(* CODESYS project mobject-converters.library
   Company: mobject
   DefaultNamespace: mobject-converters
   Version: 1.0.2
   Placeholder: mobject-converters
   Author: mobject dev team
   Title: mobject-converters

Project tree, tasks and I/O mapping:
  libraries: Tc2_System, * (Beckhoff Automation GmbH); mobject-constants-datatype-limits, 1.0.0 (mobject)
  Converters/
    BOOL_TO_/
      function TryConvert_BOOL_TO_BOOL [ST]
      function TryConvert_BOOL_TO_BYTE [ST]
      function TryConvert_BOOL_TO_DATE [ST]
      function TryConvert_BOOL_TO_Destination [ST]
      function TryConvert_BOOL_TO_DINT [ST]
      function TryConvert_BOOL_TO_DT [ST]
      function TryConvert_BOOL_TO_DWORD [ST]
      function TryConvert_BOOL_TO_INT [ST]
      function TryConvert_BOOL_TO_LINT [ST]
      function TryConvert_BOOL_TO_LREAL [ST]
      function TryConvert_BOOL_TO_LWORD [ST]
      function TryConvert_BOOL_TO_REAL [ST]
      function TryConvert_BOOL_TO_SINT [ST]
      function TryConvert_BOOL_TO_STRING [ST]
      function TryConvert_BOOL_TO_TIME [ST]
      function TryConvert_BOOL_TO_TOD [ST]
      function TryConvert_BOOL_TO_UDINT [ST]
      function TryConvert_BOOL_TO_UINT [ST]
      function TryConvert_BOOL_TO_ULINT [ST]
      function TryConvert_BOOL_TO_USINT [ST]
      function TryConvert_BOOL_TO_WORD [ST]
    BYTE_TO_/
      function TryConvert_BYTE_TO_BOOL [ST]
      function TryConvert_BYTE_TO_BYTE [ST]
      function TryConvert_BYTE_TO_DATE [ST]
      function TryConvert_BYTE_TO_Destination [ST]
      function TryConvert_BYTE_TO_DINT [ST]
      function TryConvert_BYTE_TO_DT [ST]
      function TryConvert_BYTE_TO_DWORD [ST]
      function TryConvert_BYTE_TO_INT [ST]
      function TryConvert_BYTE_TO_LINT [ST]
      function TryConvert_BYTE_TO_LREAL [ST]
      function TryConvert_BYTE_TO_LWORD [ST]
      function TryConvert_BYTE_TO_REAL [ST]
      function TryConvert_BYTE_TO_SINT [ST]
      function TryConvert_BYTE_TO_STRING [ST]
      function TryConvert_BYTE_TO_TIME [ST]
      function TryConvert_BYTE_TO_TOD [ST]
      function TryConvert_BYTE_TO_UDINT [ST]
      function TryConvert_BYTE_TO_UINT [ST]
      function TryConvert_BYTE_TO_ULINT [ST]
      function TryConvert_BYTE_TO_USINT [ST]
      function TryConvert_BYTE_TO_WORD [ST]
    DATE_TO_/
      function TryConvert_DATE_TO_BOOL [ST]
      function TryConvert_DATE_TO_BYTE [ST]
      function TryConvert_DATE_TO_DATE [ST]
      function TryConvert_DATE_TO_Destination [ST]
      function TryConvert_DATE_TO_DINT [ST]
      function TryConvert_DATE_TO_DT [ST]
      function TryConvert_DATE_TO_DWORD [ST]
      function TryConvert_DATE_TO_INT [ST]
      function TryConvert_DATE_TO_LINT [ST]
      function TryConvert_DATE_TO_LREAL [ST]
      function TryConvert_DATE_TO_LWORD [ST]
      function TryConvert_DATE_TO_REAL [ST]
      function TryConvert_DATE_TO_SINT [ST]
      function TryConvert_DATE_TO_STRING [ST]
      function TryConvert_DATE_TO_TIME [ST]
      function TryConvert_DATE_TO_TOD [ST]
      function TryConvert_DATE_TO_UDINT [ST]
      function TryConvert_DATE_TO_UINT [ST]
      function TryConvert_DATE_TO_ULINT [ST]
      function TryConvert_DATE_TO_USINT [ST]
      function TryConvert_DATE_TO_WORD [ST]
    DINT_TO_/
      function TryConvert_DINT_TO_BOOL [ST]
      function TryConvert_DINT_TO_BYTE [ST]
      function TryConvert_DINT_TO_DATE [ST]
      function TryConvert_DINT_TO_Destination [ST]
      function TryConvert_DINT_TO_DINT [ST]
      function TryConvert_DINT_TO_DT [ST]
      function TryConvert_DINT_TO_DWORD [ST]
      function TryConvert_DINT_TO_INT [ST]
      function TryConvert_DINT_TO_LINT [ST]
      function TryConvert_DINT_TO_LREAL [ST]
      function TryConvert_DINT_TO_LWORD [ST]
      function TryConvert_DINT_TO_REAL [ST]
      function TryConvert_DINT_TO_SINT [ST]
      function TryConvert_DINT_TO_STRING [ST]
      function TryConvert_DINT_TO_TIME [ST]
      function TryConvert_DINT_TO_TOD [ST]
      function TryConvert_DINT_TO_UDINT [ST]
      function TryConvert_DINT_TO_UINT [ST]
      function TryConvert_DINT_TO_ULINT [ST]
      function TryConvert_DINT_TO_USINT [ST]
      function TryConvert_DINT_TO_WORD [ST]
    DT_TO_/
      function TryConvert_DT_TO_BOOL [ST]
      function TryConvert_DT_TO_BYTE [ST]
      function TryConvert_DT_TO_DATE [ST]
      function TryConvert_DT_TO_Destination [ST]
      function TryConvert_DT_TO_DINT [ST]
      function TryConvert_DT_TO_DT [ST]
      function TryConvert_DT_TO_DWORD [ST]
      function TryConvert_DT_TO_INT [ST]
      function TryConvert_DT_TO_LINT [ST]
      function TryConvert_DT_TO_LREAL [ST]
      function TryConvert_DT_TO_LWORD [ST]
      function TryConvert_DT_TO_REAL [ST]
      function TryConvert_DT_TO_SINT [ST]
      function TryConvert_DT_TO_STRING [ST]
      function TryConvert_DT_TO_TIME [ST]
      function TryConvert_DT_TO_TOD [ST]
      function TryConvert_DT_TO_UDINT [ST]
      function TryConvert_DT_TO_UINT [ST]
      function TryConvert_DT_TO_ULINT [ST]
      function TryConvert_DT_TO_USINT [ST]
      function TryConvert_DT_TO_WORD [ST]
    DWORD_TO_/
      function TryConvert_DWORD_TO_BOOL [ST]
      function TryConvert_DWORD_TO_BYTE [ST]
      function TryConvert_DWORD_TO_DATE [ST]
      function TryConvert_DWORD_TO_Destination [ST]
      function TryConvert_DWORD_TO_DINT [ST]
      function TryConvert_DWORD_TO_DT [ST]
      function TryConvert_DWORD_TO_DWORD [ST]
      function TryConvert_DWORD_TO_INT [ST]
      function TryConvert_DWORD_TO_LINT [ST]
      function TryConvert_DWORD_TO_LREAL [ST]
      function TryConvert_DWORD_TO_LWORD [ST]
      function TryConvert_DWORD_TO_REAL [ST]
      function TryConvert_DWORD_TO_SINT [ST]
      function TryConvert_DWORD_TO_STRING [ST]
      function TryConvert_DWORD_TO_TIME [ST]
      function TryConvert_DWORD_TO_TOD [ST]
      function TryConvert_DWORD_TO_UDINT [ST]
      function TryConvert_DWORD_TO_UINT [ST]
      function TryConvert_DWORD_TO_ULINT [ST]
      function TryConvert_DWORD_TO_USINT [ST]
      function TryConvert_DWORD_TO_WORD [ST]
    INT_TO_/
      function TryConvert_INT_TO_BOOL [ST]
      function TryConvert_INT_TO_BYTE [ST]
      function TryConvert_INT_TO_DATE [ST]
      function TryConvert_INT_TO_Destination [ST]
      function TryConvert_INT_TO_DINT [ST]
      function TryConvert_INT_TO_DT [ST]
      function TryConvert_INT_TO_DWORD [ST]
      function TryConvert_INT_TO_INT [ST]
      function TryConvert_INT_TO_LINT [ST]
      function TryConvert_INT_TO_LREAL [ST]
      function TryConvert_INT_TO_LWORD [ST]
      function TryConvert_INT_TO_REAL [ST]
      function TryConvert_INT_TO_SINT [ST]
      function TryConvert_INT_TO_STRING [ST]
      function TryConvert_INT_TO_TIME [ST]
      function TryConvert_INT_TO_TOD [ST]
      function TryConvert_INT_TO_UDINT [ST]
      function TryConvert_INT_TO_UINT [ST]
      function TryConvert_INT_TO_ULINT [ST]
      function TryConvert_INT_TO_USINT [ST]
      function TryConvert_INT_TO_WORD [ST]
    LINT_TO_/
      function TryConvert_LINT_TO_BOOL [ST]
      function TryConvert_LINT_TO_BYTE [ST]
      function TryConvert_LINT_TO_DATE [ST]
      function TryConvert_LINT_TO_Destination [ST]
      function TryConvert_LINT_TO_DINT [ST]
      function TryConvert_LINT_TO_DT [ST]
      function TryConvert_LINT_TO_DWORD [ST]
      function TryConvert_LINT_TO_INT [ST]
      function TryConvert_LINT_TO_LINT [ST]
      function TryConvert_LINT_TO_LREAL [ST]
      function TryConvert_LINT_TO_LWORD [ST]
      function TryConvert_LINT_TO_REAL [ST]
      function TryConvert_LINT_TO_SINT [ST]
      function TryConvert_LINT_TO_STRING [ST]
      function TryConvert_LINT_TO_TIME [ST]
      function TryConvert_LINT_TO_TOD [ST]
      function TryConvert_LINT_TO_UDINT [ST]
      function TryConvert_LINT_TO_UINT [ST]
      function TryConvert_LINT_TO_ULINT [ST]
      function TryConvert_LINT_TO_USINT [ST]
      function TryConvert_LINT_TO_WORD [ST]
    LREAL_TO_/
      function TryConvert_LREAL_TO_BOOL [ST]
      function TryConvert_LREAL_TO_BYTE [ST]
      function TryConvert_LREAL_TO_DATE [ST]
      function TryConvert_LREAL_TO_Destination [ST]
      function TryConvert_LREAL_TO_DINT [ST]
      function TryConvert_LREAL_TO_DT [ST]
      function TryConvert_LREAL_TO_DWORD [ST]
      function TryConvert_LREAL_TO_INT [ST]
      function TryConvert_LREAL_TO_LINT [ST]
      function TryConvert_LREAL_TO_LREAL [ST]
      function TryConvert_LREAL_TO_LWORD [ST]
      function TryConvert_LREAL_TO_REAL [ST]
      function TryConvert_LREAL_TO_SINT [ST]
      function TryConvert_LREAL_TO_STRING [ST]
      function TryConvert_LREAL_TO_TIME [ST]
      function TryConvert_LREAL_TO_TOD [ST]
      function TryConvert_LREAL_TO_UDINT [ST]
      function TryConvert_LREAL_TO_UINT [ST]
      function TryConvert_LREAL_TO_ULINT [ST]
      function TryConvert_LREAL_TO_USINT [ST]
      function TryConvert_LREAL_TO_WORD [ST]
    LWORD_TO_/
      function TryConvert_LWORD_TO_BOOL [ST]
      function TryConvert_LWORD_TO_BYTE [ST]
      function TryConvert_LWORD_TO_DATE [ST]
      function TryConvert_LWORD_TO_Destination [ST]
      function TryConvert_LWORD_TO_DINT [ST]
      function TryConvert_LWORD_TO_DT [ST]
      function TryConvert_LWORD_TO_DWORD [ST]
      function TryConvert_LWORD_TO_INT [ST]
      function TryConvert_LWORD_TO_LINT [ST]
      function TryConvert_LWORD_TO_LREAL [ST]
      function TryConvert_LWORD_TO_LWORD [ST]
      function TryConvert_LWORD_TO_REAL [ST]
      function TryConvert_LWORD_TO_SINT [ST]
      function TryConvert_LWORD_TO_STRING [ST]
      function TryConvert_LWORD_TO_TIME [ST]
      function TryConvert_LWORD_TO_TOD [ST]
      function TryConvert_LWORD_TO_UDINT [ST]
      function TryConvert_LWORD_TO_UINT [ST]
      function TryConvert_LWORD_TO_ULINT [ST]
      function TryConvert_LWORD_TO_USINT [ST]
      function TryConvert_LWORD_TO_WORD [ST]
    REAL_TO_/
      function TryConvert_REAL_TO_BOOL [ST]
      function TryConvert_REAL_TO_BYTE [ST]
      function TryConvert_REAL_TO_DATE [ST]
      function TryConvert_REAL_TO_Destination [ST]
      function TryConvert_REAL_TO_DINT [ST]
      function TryConvert_REAL_TO_DT [ST]
      function TryConvert_REAL_TO_DWORD [ST]
      function TryConvert_REAL_TO_INT [ST]
      function TryConvert_REAL_TO_LINT [ST]
      function TryConvert_REAL_TO_LREAL [ST]
      function TryConvert_REAL_TO_LWORD [ST]
      function TryConvert_REAL_TO_REAL [ST]
      function TryConvert_REAL_TO_SINT [ST]
      function TryConvert_REAL_TO_STRING [ST]
      function TryConvert_REAL_TO_TIME [ST]
      function TryConvert_REAL_TO_TOD [ST]
      function TryConvert_REAL_TO_UDINT [ST]
      function TryConvert_REAL_TO_UINT [ST]
      function TryConvert_REAL_TO_ULINT [ST]
      function TryConvert_REAL_TO_USINT [ST]
      function TryConvert_REAL_TO_WORD [ST]
    SINT_TO_/
      function TryConvert_SINT_TO_BOOL [ST]
      function TryConvert_SINT_TO_BYTE [ST]
      function TryConvert_SINT_TO_DATE [ST]
      function TryConvert_SINT_TO_Destination [ST]
      function TryConvert_SINT_TO_DINT [ST]
      function TryConvert_SINT_TO_DT [ST]
      function TryConvert_SINT_TO_DWORD [ST]
      function TryConvert_SINT_TO_INT [ST]
      function TryConvert_SINT_TO_LINT [ST]
      function TryConvert_SINT_TO_LREAL [ST]
      function TryConvert_SINT_TO_LWORD [ST]
      function TryConvert_SINT_TO_REAL [ST]
      function TryConvert_SINT_TO_SINT [ST]
      function TryConvert_SINT_TO_STRING [ST]
      function TryConvert_SINT_TO_TIME [ST]
      function TryConvert_SINT_TO_TOD [ST]
      function TryConvert_SINT_TO_UDINT [ST]
      function TryConvert_SINT_TO_UINT [ST]
      function TryConvert_SINT_TO_ULINT [ST]
      function TryConvert_SINT_TO_USINT [ST]
      function TryConvert_SINT_TO_WORD [ST]
    STRING_TO_/
      function TryConvert_STRING_TO_BOOL [ST]
      function TryConvert_STRING_TO_BYTE [ST]
      function TryConvert_STRING_TO_DATE [ST]
      function TryConvert_STRING_TO_Destination [ST]
      function TryConvert_STRING_TO_DINT [ST]
      function TryConvert_STRING_TO_DT [ST]
      function TryConvert_STRING_TO_DWORD [ST]
      function TryConvert_STRING_TO_INT [ST]
      function TryConvert_STRING_TO_LINT [ST]
      function TryConvert_STRING_TO_LREAL [ST]
      function TryConvert_STRING_TO_LWORD [ST]
      function TryConvert_STRING_TO_REAL [ST]
      function TryConvert_STRING_TO_SINT [ST]
      function TryConvert_STRING_TO_STRING [ST]
      function TryConvert_STRING_TO_TIME [ST]
      function TryConvert_STRING_TO_TOD [ST]
      function TryConvert_STRING_TO_UDINT [ST]
      function TryConvert_STRING_TO_UINT [ST]
      function TryConvert_STRING_TO_ULINT [ST]
      function TryConvert_STRING_TO_USINT [ST]
      function TryConvert_STRING_TO_WORD [ST]
    TIME_TO_/
      function TryConvert_TIME_TO_BOOL [ST]
      function TryConvert_TIME_TO_BYTE [ST]
      function TryConvert_TIME_TO_DATE [ST]
      function TryConvert_TIME_TO_Destination [ST]
      function TryConvert_TIME_TO_DINT [ST]
      function TryConvert_TIME_TO_DT [ST]
      function TryConvert_TIME_TO_DWORD [ST]
      function TryConvert_TIME_TO_INT [ST]
      function TryConvert_TIME_TO_LINT [ST]
      function TryConvert_TIME_TO_LREAL [ST]
      function TryConvert_TIME_TO_LWORD [ST]
      function TryConvert_TIME_TO_REAL [ST]
      function TryConvert_TIME_TO_SINT [ST]
      function TryConvert_TIME_TO_STRING [ST]
      function TryConvert_TIME_TO_TIME [ST]
      function TryConvert_TIME_TO_TOD [ST]
      function TryConvert_TIME_TO_UDINT [ST]
      function TryConvert_TIME_TO_UINT [ST]
      function TryConvert_TIME_TO_ULINT [ST]
      function TryConvert_TIME_TO_USINT [ST]
      function TryConvert_TIME_TO_WORD [ST]
    TOD_TO_/
      function TryConvert_TOD_TO_BOOL [ST]
      function TryConvert_TOD_TO_BYTE [ST]
      function TryConvert_TOD_TO_DATE [ST]
      function TryConvert_TOD_TO_Destination [ST]
      function TryConvert_TOD_TO_DINT [ST]
      function TryConvert_TOD_TO_DT [ST]
      function TryConvert_TOD_TO_DWORD [ST]
      function TryConvert_TOD_TO_INT [ST]
      function TryConvert_TOD_TO_LINT [ST]
      function TryConvert_TOD_TO_LREAL [ST]
      function TryConvert_TOD_TO_LWORD [ST]
      function TryConvert_TOD_TO_REAL [ST]
      function TryConvert_TOD_TO_SINT [ST]
      function TryConvert_TOD_TO_STRING [ST]
      function TryConvert_TOD_TO_TIME [ST]
      function TryConvert_TOD_TO_TOD [ST]
      function TryConvert_TOD_TO_UDINT [ST]
      function TryConvert_TOD_TO_UINT [ST]
      function TryConvert_TOD_TO_ULINT [ST]
      function TryConvert_TOD_TO_USINT [ST]
      function TryConvert_TOD_TO_WORD [ST]
    UDINT_TO_/
      function TryConvert_UDINT_TO_BOOL [ST]
      function TryConvert_UDINT_TO_BYTE [ST]
      function TryConvert_UDINT_TO_DATE [ST]
      function TryConvert_UDINT_TO_Destination [ST]
      function TryConvert_UDINT_TO_DINT [ST]
      function TryConvert_UDINT_TO_DT [ST]
      function TryConvert_UDINT_TO_DWORD [ST]
      function TryConvert_UDINT_TO_INT [ST]
      function TryConvert_UDINT_TO_LINT [ST]
      function TryConvert_UDINT_TO_LREAL [ST]
      function TryConvert_UDINT_TO_LWORD [ST]
      function TryConvert_UDINT_TO_REAL [ST]
      function TryConvert_UDINT_TO_SINT [ST]
      function TryConvert_UDINT_TO_STRING [ST]
      function TryConvert_UDINT_TO_TIME [ST]
      function TryConvert_UDINT_TO_TOD [ST]
      function TryConvert_UDINT_TO_UDINT [ST]
      function TryConvert_UDINT_TO_UINT [ST]
      function TryConvert_UDINT_TO_ULINT [ST]
      function TryConvert_UDINT_TO_USINT [ST]
      function TryConvert_UDINT_TO_WORD [ST]
    UINT_TO_/
      function TryConvert_UINT_TO_BOOL [ST]
      function TryConvert_UINT_TO_BYTE [ST]
      function TryConvert_UINT_TO_DATE [ST]
      function TryConvert_UINT_TO_Destination [ST]
      function TryConvert_UINT_TO_DINT [ST]
      function TryConvert_UINT_TO_DT [ST]
      function TryConvert_UINT_TO_DWORD [ST]
      function TryConvert_UINT_TO_INT [ST]
      function TryConvert_UINT_TO_LINT [ST]
      function TryConvert_UINT_TO_LREAL [ST]
      function TryConvert_UINT_TO_LWORD [ST]
      function TryConvert_UINT_TO_REAL [ST]
      function TryConvert_UINT_TO_SINT [ST]
      function TryConvert_UINT_TO_STRING [ST]
      function TryConvert_UINT_TO_TIME [ST]
      function TryConvert_UINT_TO_TOD [ST]
      function TryConvert_UINT_TO_UDINT [ST]
      function TryConvert_UINT_TO_UINT [ST]
      function TryConvert_UINT_TO_ULINT [ST]
      function TryConvert_UINT_TO_USINT [ST]
      function TryConvert_UINT_TO_WORD [ST]
    ULINT_TO_/
      function TryConvert_ULINT_TO_BOOL [ST]
      function TryConvert_ULINT_TO_BYTE [ST]
      function TryConvert_ULINT_TO_DATE [ST]
      function TryConvert_ULINT_TO_Destination [ST]
      function TryConvert_ULINT_TO_DINT [ST]
      function TryConvert_ULINT_TO_DT [ST]
      function TryConvert_ULINT_TO_DWORD [ST]
      function TryConvert_ULINT_TO_INT [ST]
      function TryConvert_ULINT_TO_LINT [ST]
      function TryConvert_ULINT_TO_LREAL [ST]
      function TryConvert_ULINT_TO_LWORD [ST]
      function TryConvert_ULINT_TO_REAL [ST]
      function TryConvert_ULINT_TO_SINT [ST]
      function TryConvert_ULINT_TO_STRING [ST]
      function TryConvert_ULINT_TO_TIME [ST]
      function TryConvert_ULINT_TO_TOD [ST]
      function TryConvert_ULINT_TO_UDINT [ST]
      function TryConvert_ULINT_TO_UINT [ST]
      function TryConvert_ULINT_TO_ULINT [ST]
      function TryConvert_ULINT_TO_USINT [ST]
      function TryConvert_ULINT_TO_WORD [ST]
    USINT_TO_/
      function TryConvert_USINT_TO_BOOL [ST]
      function TryConvert_USINT_TO_BYTE [ST]
      function TryConvert_USINT_TO_DATE [ST]
      function TryConvert_USINT_TO_Destination [ST]
      function TryConvert_USINT_TO_DINT [ST]
      function TryConvert_USINT_TO_DT [ST]
      function TryConvert_USINT_TO_DWORD [ST]
      function TryConvert_USINT_TO_INT [ST]
      function TryConvert_USINT_TO_LINT [ST]
      function TryConvert_USINT_TO_LREAL [ST]
      function TryConvert_USINT_TO_LWORD [ST]
      function TryConvert_USINT_TO_REAL [ST]
      function TryConvert_USINT_TO_SINT [ST]
      function TryConvert_USINT_TO_STRING [ST]
      function TryConvert_USINT_TO_TIME [ST]
      function TryConvert_USINT_TO_TOD [ST]
      function TryConvert_USINT_TO_UDINT [ST]
      function TryConvert_USINT_TO_UINT [ST]
      function TryConvert_USINT_TO_ULINT [ST]
      function TryConvert_USINT_TO_USINT [ST]
      function TryConvert_USINT_TO_WORD [ST]
    WORD_TO_/
      function TryConvert_WORD_TO_BOOL [ST]
      function TryConvert_WORD_TO_BYTE [ST]
      function TryConvert_WORD_TO_DATE [ST]
      function TryConvert_WORD_TO_Destination [ST]
      function TryConvert_WORD_TO_DINT [ST]
      function TryConvert_WORD_TO_DT [ST]
      function TryConvert_WORD_TO_DWORD [ST]
      function TryConvert_WORD_TO_INT [ST]
      function TryConvert_WORD_TO_LINT [ST]
      function TryConvert_WORD_TO_LREAL [ST]
      function TryConvert_WORD_TO_LWORD [ST]
      function TryConvert_WORD_TO_REAL [ST]
      function TryConvert_WORD_TO_SINT [ST]
      function TryConvert_WORD_TO_STRING [ST]
      function TryConvert_WORD_TO_TIME [ST]
      function TryConvert_WORD_TO_TOD [ST]
      function TryConvert_WORD_TO_UDINT [ST]
      function TryConvert_WORD_TO_UINT [ST]
      function TryConvert_WORD_TO_ULINT [ST]
      function TryConvert_WORD_TO_USINT [ST]
      function TryConvert_WORD_TO_WORD [ST]
    function TryConvert_Source_TO_Destination [ST]
*)

// Converters/BOOL_TO_/TryConvert_BOOL_TO_BOOL
FUNCTION TryConvert_BOOL_TO_BOOL : BOOL
VAR_INPUT
	in : BOOL;
	out : REFERENCE TO BOOL;
END_VAR

out := in;
TryConvert_BOOL_TO_BOOL := TRUE;

END_FUNCTION

// Converters/BOOL_TO_/TryConvert_BOOL_TO_BYTE
FUNCTION TryConvert_BOOL_TO_BYTE : BOOL
VAR_INPUT
	in : BOOL;
	out : REFERENCE TO BYTE;
END_VAR

out := BOOL_TO_BYTE(in);
TryConvert_BOOL_TO_BYTE := TRUE;

END_FUNCTION

// Converters/BOOL_TO_/TryConvert_BOOL_TO_DATE
FUNCTION TryConvert_BOOL_TO_DATE : BOOL
VAR_INPUT
	in : BOOL;
	out : REFERENCE TO DATE;
END_VAR

out := BOOL_TO_DATE(in);
TryConvert_BOOL_TO_DATE := TRUE;

END_FUNCTION

// Converters/BOOL_TO_/TryConvert_BOOL_TO_Destination
FUNCTION TryConvert_BOOL_TO_Destination : BOOL
VAR_INPUT
	in : BOOL;
	out : ANY;
END_VAR
VAR
	convertResult : BOOL := FALSE;
	convertAddress : PVOID;
	_BOOL : BOOL;
	_BYTE : BYTE;
	_WORD : WORD;
	_DWORD : DWORD;
	_LWORD : LWORD;
	_SINT : SINT;
	_INT : INT;
	_DINT : DINT;
	_LINT : LINT;
	_USINT : USINT;
	_UINT : UINT;
	_UDINT : UDINT;
	_ULINT : ULINT;
	_REAL : REAL;
	_LREAL : LREAL;
	_TIME : TIME;
	_TOD : TOD;
	_DATE : DATE;
	_DT : DT;
	_STRING : STRING;
END_VAR

CASE out.TypeClass OF
	__SYSTEM.TYPE_CLASS.TYPE_BOOL:
	
	convertResult := TryConvert_BOOL_TO_BOOL(in, _BOOL);
	IF convertResult THEN
		convertAddress := ADR(_BOOL);
	END_IF
	
	__SYSTEM.TYPE_CLASS.TYPE_BYTE:
	
	convertResult := TryConvert_BOOL_TO_BYTE(in, _BYTE);
	IF convertResult THEN
		convertAddress := ADR(_BYTE);
	END_IF
	
	__SYSTEM.TYPE_CLASS.TYPE_WORD:
	
	convertResult := TryConvert_BOOL_TO_WORD(in, _WORD);
	IF convertResult THEN
		convertAddress := ADR(_WORD);
	END_IF
	
	__SYSTEM.TYPE_CLASS.TYPE_DWORD:
	
	convertResult := TryConvert_BOOL_TO_DWORD(in, _DWORD);
	IF convertResult THEN
		convertAddress := ADR(_DWORD);
	END_IF
	
	__SYSTEM.TYPE_CLASS.TYPE_LWORD:
	
	convertResult := TryConvert_BOOL_TO_LWORD(in, _LWORD);
	IF convertResult THEN
		convertAddress := ADR(_LWORD);
	END_IF
	
	__SYSTEM.TYPE_CLASS.TYPE_SINT:
	
	convertResult := TryConvert_BOOL_TO_SINT(in, _SINT);
	IF convertResult THEN
		convertAddress := ADR(_SINT);
	END_IF
	
	__SYSTEM.TYPE_CLASS.TYPE_INT:
	
	convertResult := TryConvert_BOOL_TO_INT(in, _INT);
	IF convertResult THEN
		convertAddress := ADR(_INT);
	END_IF
	
	__SYSTEM.TYPE_CLASS.TYPE_DINT:
	
	convertResult := TryConvert_BOOL_TO_DINT(in, _DINT);
	IF convertResult THEN
		convertAddress := ADR(_DINT);
	END_IF
	
	__SYSTEM.TYPE_CLASS.TYPE_LINT:
	
	convertResult := TryConvert_BOOL_TO_LINT(in, _LINT);
	IF convertResult THEN
		convertAddress := ADR(_LINT);
	END_IF
	
	__SYSTEM.TYPE_CLASS.TYPE_USINT:
	
	convertResult := TryConvert_BOOL_TO_USINT(in, _USINT);
	IF convertResult THEN
		convertAddress := ADR(_USINT);
	END_IF
	
	__SYSTEM.TYPE_CLASS.TYPE_UINT:
	
	convertResult := TryConvert_BOOL_TO_UINT(in, _UINT);
	IF convertResult THEN
		convertAddress := ADR(_UINT);
	END_IF
	
	__SYSTEM.TYPE_CLASS.TYPE_UDINT:
	
	convertResult := TryConvert_BOOL_TO_UDINT(in, _UDINT);
	IF convertResult THEN
		convertAddress := ADR(_UDINT);
	END_IF
	
	__SYSTEM.TYPE_CLASS.TYPE_ULINT:
	
	convertResult := TryConvert_BOOL_TO_ULINT(in, _ULINT);
	IF convertResult THEN
		convertAddress := ADR(_ULINT);
	END_IF
	
	__SYSTEM.TYPE_CLASS.TYPE_REAL:
	
	convertResult := TryConvert_BOOL_TO_REAL(in, _REAL);
	IF convertResult THEN
		convertAddress := ADR(_REAL);
	END_IF
	
	__SYSTEM.TYPE_CLASS.TYPE_LREAL:
	
	convertResult := TryConvert_BOOL_TO_LREAL(in, _LREAL);
	IF convertResult THEN
		convertAddress := ADR(_LREAL);
	END_IF
	
	__SYSTEM.TYPE_CLASS.TYPE_TIME:
	
	convertResult := TryConvert_BOOL_TO_TIME(in, _TIME);
	IF convertResult THEN
		convertAddress := ADR(_TIME);
	END_IF
	
	__SYSTEM.TYPE_CLASS.TYPE_TIMEOFDAY:
	
	convertResult := TryConvert_BOOL_TO_TOD(in, _TOD);
	IF convertResult THEN
		convertAddress := ADR(_TOD);
	END_IF
	
	__SYSTEM.TYPE_CLASS.TYPE_DATE:
	
	convertResult := TryConvert_BOOL_TO_DATE(in, _DATE);
	IF convertResult THEN
		convertAddress := ADR(_DATE);
	END_IF
	
	__SYSTEM.TYPE_CLASS.TYPE_DATEANDTIME:
	
	convertResult := TryConvert_BOOL_TO_DT(in, _DT);
	IF convertResult THEN
		convertAddress := ADR(_DT);
	END_IF
	
	__SYSTEM.TYPE_CLASS.TYPE_STRING:
	
	convertResult := TryConvert_BOOL_TO_STRING(in, _STRING);
	IF convertResult THEN
		convertAddress := ADR(_STRING);
	END_IF
	
END_CASE

IF convertResult THEN
	memcpy(out.pValue,convertAddress,DINT_TO_UDINT(out.diSize));
END_IF

TryConvert_BOOL_TO_Destination := convertResult;

END_FUNCTION

// Converters/BOOL_TO_/TryConvert_BOOL_TO_WORD
FUNCTION TryConvert_BOOL_TO_WORD : BOOL
VAR_INPUT
	in : BOOL;
	out : REFERENCE TO WORD;
END_VAR

out := BOOL_TO_WORD(in);
TryConvert_BOOL_TO_WORD := TRUE;

END_FUNCTION

// Converters/BOOL_TO_/TryConvert_BOOL_TO_DWORD
FUNCTION TryConvert_BOOL_TO_DWORD : BOOL
VAR_INPUT
	in : BOOL;
	out : REFERENCE TO DWORD;
END_VAR

out := BOOL_TO_DWORD(in);
TryConvert_BOOL_TO_DWORD := TRUE;

END_FUNCTION

// Converters/BOOL_TO_/TryConvert_BOOL_TO_LWORD
FUNCTION TryConvert_BOOL_TO_LWORD : BOOL
VAR_INPUT
	in : BOOL;
	out : REFERENCE TO LWORD;
END_VAR

out := BOOL_TO_LWORD(in);
TryConvert_BOOL_TO_LWORD := TRUE;

END_FUNCTION

// Converters/BOOL_TO_/TryConvert_BOOL_TO_SINT
FUNCTION TryConvert_BOOL_TO_SINT : BOOL
VAR_INPUT
	in : BOOL;
	out : REFERENCE TO SINT;
END_VAR

out := BOOL_TO_SINT(in);
TryConvert_BOOL_TO_SINT := TRUE;

END_FUNCTION

// Converters/BOOL_TO_/TryConvert_BOOL_TO_INT
FUNCTION TryConvert_BOOL_TO_INT : BOOL
VAR_INPUT
	in : BOOL;
	out : REFERENCE TO INT;
END_VAR

out := BOOL_TO_INT(in);
TryConvert_BOOL_TO_INT := TRUE;

END_FUNCTION

// Converters/BOOL_TO_/TryConvert_BOOL_TO_DINT
FUNCTION TryConvert_BOOL_TO_DINT : BOOL
VAR_INPUT
	in : BOOL;
	out : REFERENCE TO DINT;
END_VAR

out := BOOL_TO_DINT(in);
TryConvert_BOOL_TO_DINT := TRUE;

END_FUNCTION

// Converters/BOOL_TO_/TryConvert_BOOL_TO_LINT
FUNCTION TryConvert_BOOL_TO_LINT : BOOL
VAR_INPUT
	in : BOOL;
	out : REFERENCE TO LINT;
END_VAR

out := BOOL_TO_LINT(in);
TryConvert_BOOL_TO_LINT := TRUE;

END_FUNCTION

// Converters/BOOL_TO_/TryConvert_BOOL_TO_USINT
FUNCTION TryConvert_BOOL_TO_USINT : BOOL
VAR_INPUT
	in : BOOL;
	out : REFERENCE TO USINT;
END_VAR

out := BOOL_TO_USINT(in);
TryConvert_BOOL_TO_USINT := TRUE;

END_FUNCTION

// Converters/BOOL_TO_/TryConvert_BOOL_TO_UINT
FUNCTION TryConvert_BOOL_TO_UINT : BOOL
VAR_INPUT
	in : BOOL;
	out : REFERENCE TO UINT;
END_VAR

out := BOOL_TO_UINT(in);
TryConvert_BOOL_TO_UINT := TRUE;

END_FUNCTION

// Converters/BOOL_TO_/TryConvert_BOOL_TO_UDINT
FUNCTION TryConvert_BOOL_TO_UDINT : BOOL
VAR_INPUT
	in : BOOL;
	out : REFERENCE TO UDINT;
END_VAR

out := BOOL_TO_UDINT(in);
TryConvert_BOOL_TO_UDINT := TRUE;

END_FUNCTION

// Converters/BOOL_TO_/TryConvert_BOOL_TO_ULINT
FUNCTION TryConvert_BOOL_TO_ULINT : BOOL
VAR_INPUT
	in : BOOL;
	out : REFERENCE TO ULINT;
END_VAR

out := BOOL_TO_ULINT(in);
TryConvert_BOOL_TO_ULINT := TRUE;

END_FUNCTION

// Converters/BOOL_TO_/TryConvert_BOOL_TO_REAL
FUNCTION TryConvert_BOOL_TO_REAL : BOOL
VAR_INPUT
	in : BOOL;
	out : REFERENCE TO REAL;
END_VAR

out := BOOL_TO_REAL(in);
TryConvert_BOOL_TO_REAL := TRUE;

END_FUNCTION

// Converters/BOOL_TO_/TryConvert_BOOL_TO_LREAL
FUNCTION TryConvert_BOOL_TO_LREAL : BOOL
VAR_INPUT
	in : BOOL;
	out : REFERENCE TO LREAL;
END_VAR

out := BOOL_TO_LREAL(in);
TryConvert_BOOL_TO_LREAL := TRUE;

END_FUNCTION

// Converters/BOOL_TO_/TryConvert_BOOL_TO_TIME
FUNCTION TryConvert_BOOL_TO_TIME : BOOL
VAR_INPUT
	in : BOOL;
	out : REFERENCE TO TIME;
END_VAR

out := BOOL_TO_TIME(in);
TryConvert_BOOL_TO_TIME := TRUE;

END_FUNCTION

// Converters/BOOL_TO_/TryConvert_BOOL_TO_TOD
FUNCTION TryConvert_BOOL_TO_TOD : BOOL
VAR_INPUT
	in : BOOL;
	out : REFERENCE TO TOD;
END_VAR

out := BOOL_TO_TOD(in);
TryConvert_BOOL_TO_TOD := TRUE;

END_FUNCTION

// Converters/BOOL_TO_/TryConvert_BOOL_TO_DT
FUNCTION TryConvert_BOOL_TO_DT : BOOL
VAR_INPUT
	in : BOOL;
	out : REFERENCE TO DT;
END_VAR

out := BOOL_TO_DT(in);
TryConvert_BOOL_TO_DT := TRUE;

END_FUNCTION

// Converters/BOOL_TO_/TryConvert_BOOL_TO_STRING
FUNCTION TryConvert_BOOL_TO_STRING : BOOL
VAR_INPUT
	in : BOOL;
	out : REFERENCE TO STRING;
END_VAR

out := BOOL_TO_STRING(in);
TryConvert_BOOL_TO_STRING := TRUE;

END_FUNCTION

// Converters/BYTE_TO_/TryConvert_BYTE_TO_BOOL
FUNCTION TryConvert_BYTE_TO_BOOL : BOOL
VAR_INPUT
	in : BYTE;
	out : REFERENCE TO BOOL;
END_VAR

out := BYTE_TO_BOOL(in);
TryConvert_BYTE_TO_BOOL := TRUE;

END_FUNCTION

// Converters/BYTE_TO_/TryConvert_BYTE_TO_BYTE
FUNCTION TryConvert_BYTE_TO_BYTE : BOOL
VAR_INPUT
	in : BYTE;
	out : REFERENCE TO BYTE;
END_VAR

out := in;
TryConvert_BYTE_TO_BYTE := TRUE;

END_FUNCTION

// Converters/BYTE_TO_/TryConvert_BYTE_TO_DATE
FUNCTION TryConvert_BYTE_TO_DATE : BOOL
VAR_INPUT
	in : BYTE;
	out : REFERENCE TO DATE;
END_VAR

out := BYTE_TO_DATE(in);
TryConvert_BYTE_TO_DATE := TRUE;

END_FUNCTION

// Converters/BYTE_TO_/TryConvert_BYTE_TO_Destination
FUNCTION TryConvert_BYTE_TO_Destination : BOOL
VAR_INPUT
	in : BYTE;
	out : ANY;
END_VAR
VAR
	convertResult : BOOL := FALSE;
	convertAddress : PVOID;
	_BOOL : BOOL;
	_BYTE : BYTE;
	_WORD : WORD;
	_DWORD : DWORD;
	_LWORD : LWORD;
	_SINT : SINT;
	_INT : INT;
	_DINT : DINT;
	_LINT : LINT;
	_USINT : USINT;
	_UINT : UINT;
	_UDINT : UDINT;
	_ULINT : ULINT;
	_REAL : REAL;
	_LREAL : LREAL;
	_TIME : TIME;
	_TOD : TOD;
	_DATE : DATE;
	_DT : DT;
	_STRING : STRING;
END_VAR

CASE out.TypeClass OF
	__SYSTEM.TYPE_CLASS.TYPE_BOOL:
	
	convertResult := TryConvert_BYTE_TO_BOOL(in, _BOOL);
	IF convertResult THEN
		convertAddress := ADR(_BOOL);
	END_IF
	
	__SYSTEM.TYPE_CLASS.TYPE_BYTE:
	
	convertResult := TryConvert_BYTE_TO_BYTE(in, _BYTE);
	IF convertResult THEN
		convertAddress := ADR(_BYTE);
	END_IF
	
	__SYSTEM.TYPE_CLASS.TYPE_WORD:
	
	convertResult := TryConvert_BYTE_TO_WORD(in, _WORD);
	IF convertResult THEN
		convertAddress := ADR(_WORD);
	END_IF
	
	__SYSTEM.TYPE_CLASS.TYPE_DWORD:
	
	convertResult := TryConvert_BYTE_TO_DWORD(in, _DWORD);
	IF convertResult THEN
		convertAddress := ADR(_DWORD);
	END_IF
	
	__SYSTEM.TYPE_CLASS.TYPE_LWORD:
	
	convertResult := TryConvert_BYTE_TO_LWORD(in, _LWORD);
	IF convertResult THEN
		convertAddress := ADR(_LWORD);
	END_IF
	
	__SYSTEM.TYPE_CLASS.TYPE_SINT:
	
	convertResult := TryConvert_BYTE_TO_SINT(in, _SINT);
	IF convertResult THEN
		convertAddress := ADR(_SINT);
	END_IF
	
	__SYSTEM.TYPE_CLASS.TYPE_INT:
	
	convertResult := TryConvert_BYTE_TO_INT(in, _INT);
	IF convertResult THEN
		convertAddress := ADR(_INT);
	END_IF
	
	__SYSTEM.TYPE_CLASS.TYPE_DINT:
	
	convertResult := TryConvert_BYTE_TO_DINT(in, _DINT);
	IF convertResult THEN
		convertAddress := ADR(_DINT);
	END_IF
	
	__SYSTEM.TYPE_CLASS.TYPE_LINT:
	
	convertResult := TryConvert_BYTE_TO_LINT(in, _LINT);
	IF convertResult THEN
		convertAddress := ADR(_LINT);
	END_IF
	
	__SYSTEM.TYPE_CLASS.TYPE_USINT:
	
	convertResult := TryConvert_BYTE_TO_USINT(in, _USINT);
	IF convertResult THEN
		convertAddress := ADR(_USINT);
	END_IF
	
	__SYSTEM.TYPE_CLASS.TYPE_UINT:
	
	convertResult := TryConvert_BYTE_TO_UINT(in, _UINT);
	IF convertResult THEN
		convertAddress := ADR(_UINT);
	END_IF
	
	__SYSTEM.TYPE_CLASS.TYPE_UDINT:
	
	convertResult := TryConvert_BYTE_TO_UDINT(in, _UDINT);
	IF convertResult THEN
		convertAddress := ADR(_UDINT);
	END_IF
	
	__SYSTEM.TYPE_CLASS.TYPE_ULINT:
	
	convertResult := TryConvert_BYTE_TO_ULINT(in, _ULINT);
	IF convertResult THEN
		convertAddress := ADR(_ULINT);
	END_IF
	
	__SYSTEM.TYPE_CLASS.TYPE_REAL:
	
	convertResult := TryConvert_BYTE_TO_REAL(in, _REAL);
	IF convertResult THEN
		convertAddress := ADR(_REAL);
	END_IF
	
	__SYSTEM.TYPE_CLASS.TYPE_LREAL:
	
	convertResult := TryConvert_BYTE_TO_LREAL(in, _LREAL);
	IF convertResult THEN
		convertAddress := ADR(_LREAL);
	END_IF
	
	__SYSTEM.TYPE_CLASS.TYPE_TIME:
	
	convertResult := TryConvert_BYTE_TO_TIME(in, _TIME);
	IF convertResult THEN
		convertAddress := ADR(_TIME);
	END_IF
	
	__SYSTEM.TYPE_CLASS.TYPE_TIMEOFDAY:
	
	convertResult := TryConvert_BYTE_TO_TOD(in, _TOD);
	IF convertResult THEN
		convertAddress := ADR(_TOD);
	END_IF
	
	__SYSTEM.TYPE_CLASS.TYPE_DATE:
	
	convertResult := TryConvert_BYTE_TO_DATE(in, _DATE);
	IF convertResult THEN
		convertAddress := ADR(_DATE);
	END_IF
	
	__SYSTEM.TYPE_CLASS.TYPE_DATEANDTIME:
	
	convertResult := TryConvert_BYTE_TO_DT(in, _DT);
	IF convertResult THEN
		convertAddress := ADR(_DT);
	END_IF
	
	__SYSTEM.TYPE_CLASS.TYPE_STRING:
	
	convertResult := TryConvert_BYTE_TO_STRING(in, _STRING);
	IF convertResult THEN
		convertAddress := ADR(_STRING);
	END_IF
	
END_CASE

IF convertResult THEN
	memcpy(out.pValue,convertAddress,DINT_TO_UDINT(out.diSize));
END_IF

TryConvert_BYTE_TO_Destination := convertResult;

END_FUNCTION

// Converters/BYTE_TO_/TryConvert_BYTE_TO_WORD
FUNCTION TryConvert_BYTE_TO_WORD : BOOL
VAR_INPUT
	in : BYTE;
	out : REFERENCE TO WORD;
END_VAR

out := BYTE_TO_WORD(in);
TryConvert_BYTE_TO_WORD := TRUE;

END_FUNCTION

// Converters/BYTE_TO_/TryConvert_BYTE_TO_DWORD
FUNCTION TryConvert_BYTE_TO_DWORD : BOOL
VAR_INPUT
	in : BYTE;
	out : REFERENCE TO DWORD;
END_VAR

out := BYTE_TO_DWORD(in);
TryConvert_BYTE_TO_DWORD := TRUE;

END_FUNCTION

// Converters/BYTE_TO_/TryConvert_BYTE_TO_LWORD
FUNCTION TryConvert_BYTE_TO_LWORD : BOOL
VAR_INPUT
	in : BYTE;
	out : REFERENCE TO LWORD;
END_VAR

out := BYTE_TO_LWORD(in);
TryConvert_BYTE_TO_LWORD := TRUE;

END_FUNCTION

// Converters/BYTE_TO_/TryConvert_BYTE_TO_SINT
FUNCTION TryConvert_BYTE_TO_SINT : BOOL
VAR_INPUT
	in : BYTE;
	out : REFERENCE TO SINT;
END_VAR

IF in > DatatypeLimits.MAX_VALUE_OF_BYTE_WHICH_CAN_BE_HELD_IN_A_SINT THEN
	RETURN;
END_IF

out := BYTE_TO_SINT(in);
TryConvert_BYTE_TO_SINT := TRUE;

END_FUNCTION

// Converters/BYTE_TO_/TryConvert_BYTE_TO_INT
FUNCTION TryConvert_BYTE_TO_INT : BOOL
VAR_INPUT
	in : BYTE;
	out : REFERENCE TO INT;
END_VAR

out := BYTE_TO_INT(in);
TryConvert_BYTE_TO_INT := TRUE;

END_FUNCTION

// Converters/BYTE_TO_/TryConvert_BYTE_TO_DINT
FUNCTION TryConvert_BYTE_TO_DINT : BOOL
VAR_INPUT
	in : BYTE;
	out : REFERENCE TO DINT;
END_VAR

out := BYTE_TO_DINT(in);
TryConvert_BYTE_TO_DINT := TRUE;

END_FUNCTION

// Converters/BYTE_TO_/TryConvert_BYTE_TO_LINT
FUNCTION TryConvert_BYTE_TO_LINT : BOOL
VAR_INPUT
	in : BYTE;
	out : REFERENCE TO LINT;
END_VAR

out := BYTE_TO_LINT(in);
TryConvert_BYTE_TO_LINT := TRUE;

END_FUNCTION

// Converters/BYTE_TO_/TryConvert_BYTE_TO_USINT
FUNCTION TryConvert_BYTE_TO_USINT : BOOL
VAR_INPUT
	in : BYTE;
	out : REFERENCE TO USINT;
END_VAR

out := BYTE_TO_USINT(in);
TryConvert_BYTE_TO_USINT := TRUE;

END_FUNCTION

// Converters/BYTE_TO_/TryConvert_BYTE_TO_UINT
FUNCTION TryConvert_BYTE_TO_UINT : BOOL
VAR_INPUT
	in : BYTE;
	out : REFERENCE TO UINT;
END_VAR

out := BYTE_TO_UINT(in);
TryConvert_BYTE_TO_UINT := TRUE;

END_FUNCTION

// Converters/BYTE_TO_/TryConvert_BYTE_TO_UDINT
FUNCTION TryConvert_BYTE_TO_UDINT : BOOL
VAR_INPUT
	in : BYTE;
	out : REFERENCE TO UDINT;
END_VAR

out := BYTE_TO_UDINT(in);
TryConvert_BYTE_TO_UDINT := TRUE;

END_FUNCTION

// Converters/BYTE_TO_/TryConvert_BYTE_TO_ULINT
FUNCTION TryConvert_BYTE_TO_ULINT : BOOL
VAR_INPUT
	in : BYTE;
	out : REFERENCE TO ULINT;
END_VAR

out := BYTE_TO_ULINT(in);
TryConvert_BYTE_TO_ULINT := TRUE;

END_FUNCTION

// Converters/BYTE_TO_/TryConvert_BYTE_TO_REAL
FUNCTION TryConvert_BYTE_TO_REAL : BOOL
VAR_INPUT
	in : BYTE;
	out : REFERENCE TO REAL;
END_VAR

out := BYTE_TO_REAL(in);
TryConvert_BYTE_TO_REAL := TRUE;

END_FUNCTION

// Converters/BYTE_TO_/TryConvert_BYTE_TO_LREAL
FUNCTION TryConvert_BYTE_TO_LREAL : BOOL
VAR_INPUT
	in : BYTE;
	out : REFERENCE TO LREAL;
END_VAR

out := BYTE_TO_LREAL(in);
TryConvert_BYTE_TO_LREAL := TRUE;

END_FUNCTION

// Converters/BYTE_TO_/TryConvert_BYTE_TO_TIME
FUNCTION TryConvert_BYTE_TO_TIME : BOOL
VAR_INPUT
	in : BYTE;
	out : REFERENCE TO TIME;
END_VAR

out := BYTE_TO_TIME(in);
TryConvert_BYTE_TO_TIME := TRUE;

END_FUNCTION

// Converters/BYTE_TO_/TryConvert_BYTE_TO_TOD
FUNCTION TryConvert_BYTE_TO_TOD : BOOL
VAR_INPUT
	in : BYTE;
	out : REFERENCE TO TOD;
END_VAR

out := BYTE_TO_TOD(in);
TryConvert_BYTE_TO_TOD := TRUE;

END_FUNCTION

// Converters/BYTE_TO_/TryConvert_BYTE_TO_DT
FUNCTION TryConvert_BYTE_TO_DT : BOOL
VAR_INPUT
	in : BYTE;
	out : REFERENCE TO DT;
END_VAR

out := BYTE_TO_DT(in);
TryConvert_BYTE_TO_DT := TRUE;

END_FUNCTION

// Converters/BYTE_TO_/TryConvert_BYTE_TO_STRING
FUNCTION TryConvert_BYTE_TO_STRING : BOOL
VAR_INPUT
	in : BYTE;
	out : REFERENCE TO STRING;
END_VAR

out := BYTE_TO_STRING(in);
TryConvert_BYTE_TO_STRING := TRUE;

END_FUNCTION

// Converters/DATE_TO_/TryConvert_DATE_TO_BOOL
FUNCTION TryConvert_DATE_TO_BOOL : BOOL
VAR_INPUT
	in : DATE;
	out : REFERENCE TO BOOL;
END_VAR

out := DATE_TO_BOOL(in);
TryConvert_DATE_TO_BOOL := TRUE;

END_FUNCTION

// Converters/DATE_TO_/TryConvert_DATE_TO_BYTE
FUNCTION TryConvert_DATE_TO_BYTE : BOOL
VAR_INPUT
	in : DATE;
	out : REFERENCE TO BYTE;
END_VAR

IF in > DatatypeLimits.MAX_VALUE_OF_DATE_WHICH_CAN_BE_HELD_IN_A_BYTE THEN
	RETURN;
END_IF

out := DATE_TO_BYTE(in);
TryConvert_DATE_TO_BYTE := TRUE;

END_FUNCTION

// Converters/DATE_TO_/TryConvert_DATE_TO_DATE
FUNCTION TryConvert_DATE_TO_DATE : BOOL
VAR_INPUT
	in : DATE;
	out : REFERENCE TO DATE;
END_VAR

out := in;
TryConvert_DATE_TO_DATE := TRUE;

END_FUNCTION

// Converters/DATE_TO_/TryConvert_DATE_TO_Destination
FUNCTION TryConvert_DATE_TO_Destination : BOOL
VAR_INPUT
	in : DATE;
	out : ANY;
END_VAR
VAR
	convertResult : BOOL := FALSE;
	convertAddress : PVOID;
	_BOOL : BOOL;
	_BYTE : BYTE;
	_WORD : WORD;
	_DWORD : DWORD;
	_LWORD : LWORD;
	_SINT : SINT;
	_INT : INT;
	_DINT : DINT;
	_LINT : LINT;
	_USINT : USINT;
	_UINT : UINT;
	_UDINT : UDINT;
	_ULINT : ULINT;
	_REAL : REAL;
	_LREAL : LREAL;
	_TIME : TIME;
	_TOD : TOD;
	_DATE : DATE;
	_DT : DT;
	_STRING : STRING;
END_VAR

CASE out.TypeClass OF
	__SYSTEM.TYPE_CLASS.TYPE_BOOL:
	
	convertResult := TryConvert_DATE_TO_BOOL(in, _BOOL);
	IF convertResult THEN
		convertAddress := ADR(_BOOL);
	END_IF
	
	__SYSTEM.TYPE_CLASS.TYPE_BYTE:
	
	convertResult := TryConvert_DATE_TO_BYTE(in, _BYTE);
	IF convertResult THEN
		convertAddress := ADR(_BYTE);
	END_IF
	
	__SYSTEM.TYPE_CLASS.TYPE_WORD:
	
	convertResult := TryConvert_DATE_TO_WORD(in, _WORD);
	IF convertResult THEN
		convertAddress := ADR(_WORD);
	END_IF
	
	__SYSTEM.TYPE_CLASS.TYPE_DWORD:
	
	convertResult := TryConvert_DATE_TO_DWORD(in, _DWORD);
	IF convertResult THEN
		convertAddress := ADR(_DWORD);
	END_IF
	
	__SYSTEM.TYPE_CLASS.TYPE_LWORD:
	
	convertResult := TryConvert_DATE_TO_LWORD(in, _LWORD);
	IF convertResult THEN
		convertAddress := ADR(_LWORD);
	END_IF
	
	__SYSTEM.TYPE_CLASS.TYPE_SINT:
	
	convertResult := TryConvert_DATE_TO_SINT(in, _SINT);
	IF convertResult THEN
		convertAddress := ADR(_SINT);
	END_IF
	
	__SYSTEM.TYPE_CLASS.TYPE_INT:
	
	convertResult := TryConvert_DATE_TO_INT(in, _INT);
	IF convertResult THEN
		convertAddress := ADR(_INT);
	END_IF
	
	__SYSTEM.TYPE_CLASS.TYPE_DINT:
	
	convertResult := TryConvert_DATE_TO_DINT(in, _DINT);
	IF convertResult THEN
		convertAddress := ADR(_DINT);
	END_IF
	
	__SYSTEM.TYPE_CLASS.TYPE_LINT:
	
	convertResult := TryConvert_DATE_TO_LINT(in, _LINT);
	IF convertResult THEN
		convertAddress := ADR(_LINT);
	END_IF
	
	__SYSTEM.TYPE_CLASS.TYPE_USINT:
	
	convertResult := TryConvert_DATE_TO_USINT(in, _USINT);
	IF convertResult THEN
		convertAddress := ADR(_USINT);
	END_IF
	
	__SYSTEM.TYPE_CLASS.TYPE_UINT:
	
	convertResult := TryConvert_DATE_TO_UINT(in, _UINT);
	IF convertResult THEN
		convertAddress := ADR(_UINT);
	END_IF
	
	__SYSTEM.TYPE_CLASS.TYPE_UDINT:
	
	convertResult := TryConvert_DATE_TO_UDINT(in, _UDINT);
	IF convertResult THEN
		convertAddress := ADR(_UDINT);
	END_IF
	
	__SYSTEM.TYPE_CLASS.TYPE_ULINT:
	
	convertResult := TryConvert_DATE_TO_ULINT(in, _ULINT);
	IF convertResult THEN
		convertAddress := ADR(_ULINT);
	END_IF
	
	__SYSTEM.TYPE_CLASS.TYPE_REAL:
	
	convertResult := TryConvert_DATE_TO_REAL(in, _REAL);
	IF convertResult THEN
		convertAddress := ADR(_REAL);
	END_IF
	
	__SYSTEM.TYPE_CLASS.TYPE_LREAL:
	
	convertResult := TryConvert_DATE_TO_LREAL(in, _LREAL);
	IF convertResult THEN
		convertAddress := ADR(_LREAL);
	END_IF
	
	__SYSTEM.TYPE_CLASS.TYPE_TIME:
	
	convertResult := TryConvert_DATE_TO_TIME(in, _TIME);
	IF convertResult THEN
		convertAddress := ADR(_TIME);
	END_IF
	
	__SYSTEM.TYPE_CLASS.TYPE_TIMEOFDAY:
	
	convertResult := TryConvert_DATE_TO_TOD(in, _TOD);
	IF convertResult THEN
		convertAddress := ADR(_TOD);
	END_IF
	
	__SYSTEM.TYPE_CLASS.TYPE_DATE:
	
	convertResult := TryConvert_DATE_TO_DATE(in, _DATE);
	IF convertResult THEN
		convertAddress := ADR(_DATE);
	END_IF
	
	__SYSTEM.TYPE_CLASS.TYPE_DATEANDTIME:
	
	convertResult := TryConvert_DATE_TO_DT(in, _DT);
	IF convertResult THEN
		convertAddress := ADR(_DT);
	END_IF
	
	__SYSTEM.TYPE_CLASS.TYPE_STRING:
	
	convertResult := TryConvert_DATE_TO_STRING(in, _STRING);
	IF convertResult THEN
		convertAddress := ADR(_STRING);
	END_IF
	
END_CASE

IF convertResult THEN
	memcpy(out.pValue,convertAddress,DINT_TO_UDINT(out.diSize));
END_IF

TryConvert_DATE_TO_Destination := convertResult;

END_FUNCTION

// Converters/DATE_TO_/TryConvert_DATE_TO_WORD
FUNCTION TryConvert_DATE_TO_WORD : BOOL
VAR_INPUT
	in : DATE;
	out : REFERENCE TO WORD;
END_VAR

IF in > DatatypeLimits.MAX_VALUE_OF_DATE_WHICH_CAN_BE_HELD_IN_A_WORD THEN
	RETURN;
END_IF

out := DATE_TO_WORD(in);
TryConvert_DATE_TO_WORD := TRUE;

END_FUNCTION

// Converters/DATE_TO_/TryConvert_DATE_TO_DWORD
FUNCTION TryConvert_DATE_TO_DWORD : BOOL
VAR_INPUT
	in : DATE;
	out : REFERENCE TO DWORD;
END_VAR

out := DATE_TO_DWORD(in);
TryConvert_DATE_TO_DWORD := TRUE;

END_FUNCTION

// Converters/DATE_TO_/TryConvert_DATE_TO_LWORD
FUNCTION TryConvert_DATE_TO_LWORD : BOOL
VAR_INPUT
	in : DATE;
	out : REFERENCE TO LWORD;
END_VAR

out := DATE_TO_LWORD(in);
TryConvert_DATE_TO_LWORD := TRUE;

END_FUNCTION

// Converters/DATE_TO_/TryConvert_DATE_TO_SINT
FUNCTION TryConvert_DATE_TO_SINT : BOOL
VAR_INPUT
	in : DATE;
	out : REFERENCE TO SINT;
END_VAR

IF in > DatatypeLimits.MAX_VALUE_OF_DATE_WHICH_CAN_BE_HELD_IN_A_SINT THEN
	RETURN;
END_IF

out := DATE_TO_SINT(in);
TryConvert_DATE_TO_SINT := TRUE;

END_FUNCTION

// Converters/DATE_TO_/TryConvert_DATE_TO_INT
FUNCTION TryConvert_DATE_TO_INT : BOOL
VAR_INPUT
	in : DATE;
	out : REFERENCE TO INT;
END_VAR

IF in > DatatypeLimits.MAX_VALUE_OF_DATE_WHICH_CAN_BE_HELD_IN_A_INT THEN
	RETURN;
END_IF

out := DATE_TO_INT(in);
TryConvert_DATE_TO_INT := TRUE;

END_FUNCTION

// Converters/DATE_TO_/TryConvert_DATE_TO_DINT
FUNCTION TryConvert_DATE_TO_DINT : BOOL
VAR_INPUT
	in : DATE;
	out : REFERENCE TO DINT;
END_VAR

IF in > DatatypeLimits.MAX_VALUE_OF_DATE_WHICH_CAN_BE_HELD_IN_A_DINT THEN
	RETURN;
END_IF

out := DATE_TO_DINT(in);
TryConvert_DATE_TO_DINT := TRUE;

END_FUNCTION

// Converters/DATE_TO_/TryConvert_DATE_TO_LINT
FUNCTION TryConvert_DATE_TO_LINT : BOOL
VAR_INPUT
	in : DATE;
	out : REFERENCE TO LINT;
END_VAR

out := DATE_TO_LINT(in);
TryConvert_DATE_TO_LINT := TRUE;

END_FUNCTION

// Converters/DATE_TO_/TryConvert_DATE_TO_USINT
FUNCTION TryConvert_DATE_TO_USINT : BOOL
VAR_INPUT
	in : DATE;
	out : REFERENCE TO USINT;
END_VAR

IF in > DatatypeLimits.MAX_VALUE_OF_DATE_WHICH_CAN_BE_HELD_IN_A_USINT THEN
	RETURN;
END_IF

out := DATE_TO_USINT(in);
TryConvert_DATE_TO_USINT := TRUE;

END_FUNCTION

// Converters/DATE_TO_/TryConvert_DATE_TO_UINT
FUNCTION TryConvert_DATE_TO_UINT : BOOL
VAR_INPUT
	in : DATE;
	out : REFERENCE TO UINT;
END_VAR

IF in > DatatypeLimits.MAX_VALUE_OF_DATE_WHICH_CAN_BE_HELD_IN_A_UINT THEN
	RETURN;
END_IF

out := DATE_TO_UINT(in);
TryConvert_DATE_TO_UINT := TRUE;

END_FUNCTION

// Converters/DATE_TO_/TryConvert_DATE_TO_UDINT
FUNCTION TryConvert_DATE_TO_UDINT : BOOL
VAR_INPUT
	in : DATE;
	out : REFERENCE TO UDINT;
END_VAR

out := DATE_TO_UDINT(in);
TryConvert_DATE_TO_UDINT := TRUE;

END_FUNCTION

// Converters/DATE_TO_/TryConvert_DATE_TO_ULINT
FUNCTION TryConvert_DATE_TO_ULINT : BOOL
VAR_INPUT
	in : DATE;
	out : REFERENCE TO ULINT;
END_VAR

out := DATE_TO_ULINT(in);
TryConvert_DATE_TO_ULINT := TRUE;

END_FUNCTION

// Converters/DATE_TO_/TryConvert_DATE_TO_REAL
FUNCTION TryConvert_DATE_TO_REAL : BOOL
VAR_INPUT
	in : DATE;
	out : REFERENCE TO REAL;
END_VAR

out := DATE_TO_REAL(in);
TryConvert_DATE_TO_REAL := TRUE;

END_FUNCTION

// Converters/DATE_TO_/TryConvert_DATE_TO_LREAL
FUNCTION TryConvert_DATE_TO_LREAL : BOOL
VAR_INPUT
	in : DATE;
	out : REFERENCE TO LREAL;
END_VAR

out := DATE_TO_LREAL(in);
TryConvert_DATE_TO_LREAL := TRUE;

END_FUNCTION

// Converters/DATE_TO_/TryConvert_DATE_TO_TIME
FUNCTION TryConvert_DATE_TO_TIME : BOOL
VAR_INPUT
	in : DATE;
	out : REFERENCE TO TIME;
END_VAR

IF in > DatatypeLimits.MAX_VALUE_OF_DATE_WHICH_CAN_BE_HELD_IN_A_TIME THEN
	RETURN;
END_IF

out := DATE_TO_TIME(in);
TryConvert_DATE_TO_TIME := TRUE;

END_FUNCTION

// Converters/DATE_TO_/TryConvert_DATE_TO_TOD
FUNCTION TryConvert_DATE_TO_TOD : BOOL
VAR_INPUT
	in : DATE;
	out : REFERENCE TO TOD;
END_VAR

IF in > DatatypeLimits.MAX_VALUE_OF_DATE_WHICH_CAN_BE_HELD_IN_A_TOD THEN
	RETURN;
END_IF

out := DATE_TO_TOD(in);
TryConvert_DATE_TO_TOD := TRUE;

END_FUNCTION

// Converters/DATE_TO_/TryConvert_DATE_TO_DT
FUNCTION TryConvert_DATE_TO_DT : BOOL
VAR_INPUT
	in : DATE;
	out : REFERENCE TO DT;
END_VAR

IF in > DatatypeLimits.MAX_VALUE_OF_DATE_WHICH_CAN_BE_HELD_IN_A_DT THEN
	RETURN;
END_IF

out := DATE_TO_DT(in);
TryConvert_DATE_TO_DT := TRUE;

END_FUNCTION

// Converters/DATE_TO_/TryConvert_DATE_TO_STRING
FUNCTION TryConvert_DATE_TO_STRING : BOOL
VAR_INPUT
	in : DATE;
	out : REFERENCE TO STRING;
END_VAR

out := DATE_TO_STRING(in);
TryConvert_DATE_TO_STRING := TRUE;

END_FUNCTION

// Converters/DINT_TO_/TryConvert_DINT_TO_BOOL
FUNCTION TryConvert_DINT_TO_BOOL : BOOL
VAR_INPUT
	in : DINT;
	out : REFERENCE TO BOOL;
END_VAR

out := DINT_TO_BOOL(in);
TryConvert_DINT_TO_BOOL := TRUE;

END_FUNCTION

// Converters/DINT_TO_/TryConvert_DINT_TO_BYTE
FUNCTION TryConvert_DINT_TO_BYTE : BOOL
VAR_INPUT
	in : DINT;
	out : REFERENCE TO BYTE;
END_VAR

IF in > DatatypeLimits.MAX_VALUE_OF_DINT_WHICH_CAN_BE_HELD_IN_A_BYTE THEN
	RETURN;
END_IF

IF in < DatatypeLimits.MIN_VALUE_OF_DINT_WHICH_CAN_BE_HELD_IN_A_BYTE THEN
	RETURN;
END_IF

out := DINT_TO_BYTE(in);
TryConvert_DINT_TO_BYTE := TRUE;

END_FUNCTION

// Converters/DINT_TO_/TryConvert_DINT_TO_DATE
FUNCTION TryConvert_DINT_TO_DATE : BOOL
VAR_INPUT
	in : DINT;
	out : REFERENCE TO DATE;
END_VAR

IF in < DatatypeLimits.MIN_VALUE_OF_DINT_WHICH_CAN_BE_HELD_IN_A_DATE THEN
	RETURN;
END_IF

out := DINT_TO_DATE(in);
TryConvert_DINT_TO_DATE := TRUE;

END_FUNCTION

// Converters/DINT_TO_/TryConvert_DINT_TO_Destination
FUNCTION TryConvert_DINT_TO_Destination : BOOL
VAR_INPUT
	in : DINT;
	out : ANY;
END_VAR
VAR
	convertResult : BOOL := FALSE;
	convertAddress : PVOID;
	_BOOL : BOOL;
	_BYTE : BYTE;
	_WORD : WORD;
	_DWORD : DWORD;
	_LWORD : LWORD;
	_SINT : SINT;
	_INT : INT;
	_DINT : DINT;
	_LINT : LINT;
	_USINT : USINT;
	_UINT : UINT;
	_UDINT : UDINT;
	_ULINT : ULINT;
	_REAL : REAL;
	_LREAL : LREAL;
	_TIME : TIME;
	_TOD : TOD;
	_DATE : DATE;
	_DT : DT;
	_STRING : STRING;
END_VAR

CASE out.TypeClass OF
	__SYSTEM.TYPE_CLASS.TYPE_BOOL:
	
	convertResult := TryConvert_DINT_TO_BOOL(in, _BOOL);
	IF convertResult THEN
		convertAddress := ADR(_BOOL);
	END_IF
	
	__SYSTEM.TYPE_CLASS.TYPE_BYTE:
	
	convertResult := TryConvert_DINT_TO_BYTE(in, _BYTE);
	IF convertResult THEN
		convertAddress := ADR(_BYTE);
	END_IF
	
	__SYSTEM.TYPE_CLASS.TYPE_WORD:
	
	convertResult := TryConvert_DINT_TO_WORD(in, _WORD);
	IF convertResult THEN
		convertAddress := ADR(_WORD);
	END_IF
	
	__SYSTEM.TYPE_CLASS.TYPE_DWORD:
	
	convertResult := TryConvert_DINT_TO_DWORD(in, _DWORD);
	IF convertResult THEN
		convertAddress := ADR(_DWORD);
	END_IF
	
	__SYSTEM.TYPE_CLASS.TYPE_LWORD:
	
	convertResult := TryConvert_DINT_TO_LWORD(in, _LWORD);
	IF convertResult THEN
		convertAddress := ADR(_LWORD);
	END_IF
	
	__SYSTEM.TYPE_CLASS.TYPE_SINT:
	
	convertResult := TryConvert_DINT_TO_SINT(in, _SINT);
	IF convertResult THEN
		convertAddress := ADR(_SINT);
	END_IF
	
	__SYSTEM.TYPE_CLASS.TYPE_INT:
	
	convertResult := TryConvert_DINT_TO_INT(in, _INT);
	IF convertResult THEN
		convertAddress := ADR(_INT);
	END_IF
	
	__SYSTEM.TYPE_CLASS.TYPE_DINT:
	
	convertResult := TryConvert_DINT_TO_DINT(in, _DINT);
	IF convertResult THEN
		convertAddress := ADR(_DINT);
	END_IF
	
	__SYSTEM.TYPE_CLASS.TYPE_LINT:
	
	convertResult := TryConvert_DINT_TO_LINT(in, _LINT);
	IF convertResult THEN
		convertAddress := ADR(_LINT);
	END_IF
	
	__SYSTEM.TYPE_CLASS.TYPE_USINT:
	
	convertResult := TryConvert_DINT_TO_USINT(in, _USINT);
	IF convertResult THEN
		convertAddress := ADR(_USINT);
	END_IF
	
	__SYSTEM.TYPE_CLASS.TYPE_UINT:
	
	convertResult := TryConvert_DINT_TO_UINT(in, _UINT);
	IF convertResult THEN
		convertAddress := ADR(_UINT);
	END_IF
	
	__SYSTEM.TYPE_CLASS.TYPE_UDINT:
	
	convertResult := TryConvert_DINT_TO_UDINT(in, _UDINT);
	IF convertResult THEN
		convertAddress := ADR(_UDINT);
	END_IF
	
	__SYSTEM.TYPE_CLASS.TYPE_ULINT:
	
	convertResult := TryConvert_DINT_TO_ULINT(in, _ULINT);
	IF convertResult THEN
		convertAddress := ADR(_ULINT);
	END_IF
	
	__SYSTEM.TYPE_CLASS.TYPE_REAL:
	
	convertResult := TryConvert_DINT_TO_REAL(in, _REAL);
	IF convertResult THEN
		convertAddress := ADR(_REAL);
	END_IF
	
	__SYSTEM.TYPE_CLASS.TYPE_LREAL:
	
	convertResult := TryConvert_DINT_TO_LREAL(in, _LREAL);
	IF convertResult THEN
		convertAddress := ADR(_LREAL);
	END_IF
	
	__SYSTEM.TYPE_CLASS.TYPE_TIME:
	
	convertResult := TryConvert_DINT_TO_TIME(in, _TIME);
	IF convertResult THEN
		convertAddress := ADR(_TIME);
	END_IF
	
	__SYSTEM.TYPE_CLASS.TYPE_TIMEOFDAY:
	
	convertResult := TryConvert_DINT_TO_TOD(in, _TOD);
	IF convertResult THEN
		convertAddress := ADR(_TOD);
	END_IF
	
	__SYSTEM.TYPE_CLASS.TYPE_DATE:
	
	convertResult := TryConvert_DINT_TO_DATE(in, _DATE);
	IF convertResult THEN
		convertAddress := ADR(_DATE);
	END_IF
	
	__SYSTEM.TYPE_CLASS.TYPE_DATEANDTIME:
	
	convertResult := TryConvert_DINT_TO_DT(in, _DT);
	IF convertResult THEN
		convertAddress := ADR(_DT);
	END_IF
	
	__SYSTEM.TYPE_CLASS.TYPE_STRING:
	
	convertResult := TryConvert_DINT_TO_STRING(in, _STRING);
	IF convertResult THEN
		convertAddress := ADR(_STRING);
	END_IF
	
END_CASE

IF convertResult THEN
	memcpy(out.pValue,convertAddress,DINT_TO_UDINT(out.diSize));
END_IF

TryConvert_DINT_TO_Destination := convertResult;

END_FUNCTION

// Converters/DINT_TO_/TryConvert_DINT_TO_WORD
FUNCTION TryConvert_DINT_TO_WORD : BOOL
VAR_INPUT
	in : DINT;
	out : REFERENCE TO WORD;
END_VAR

IF in > DatatypeLimits.MAX_VALUE_OF_DINT_WHICH_CAN_BE_HELD_IN_A_WORD THEN
	RETURN;
END_IF

IF in < DatatypeLimits.MIN_VALUE_OF_DINT_WHICH_CAN_BE_HELD_IN_A_WORD THEN
	RETURN;
END_IF

out := DINT_TO_WORD(in);
TryConvert_DINT_TO_WORD := TRUE;

END_FUNCTION

// Converters/DINT_TO_/TryConvert_DINT_TO_DWORD
FUNCTION TryConvert_DINT_TO_DWORD : BOOL
VAR_INPUT
	in : DINT;
	out : REFERENCE TO DWORD;
END_VAR

IF in < DatatypeLimits.MIN_VALUE_OF_DINT_WHICH_CAN_BE_HELD_IN_A_DWORD THEN
	RETURN;
END_IF

out := DINT_TO_DWORD(in);
TryConvert_DINT_TO_DWORD := TRUE;

END_FUNCTION

// Converters/DINT_TO_/TryConvert_DINT_TO_LWORD
FUNCTION TryConvert_DINT_TO_LWORD : BOOL
VAR_INPUT
	in : DINT;
	out : REFERENCE TO LWORD;
END_VAR

IF in < DatatypeLimits.MIN_VALUE_OF_DINT_WHICH_CAN_BE_HELD_IN_A_LWORD THEN
	RETURN;
END_IF

out := DINT_TO_LWORD(in);
TryConvert_DINT_TO_LWORD := TRUE;

END_FUNCTION

// Converters/DINT_TO_/TryConvert_DINT_TO_SINT
FUNCTION TryConvert_DINT_TO_SINT : BOOL
VAR_INPUT
	in : DINT;
	out : REFERENCE TO SINT;
END_VAR

IF in > DatatypeLimits.MAX_VALUE_OF_DINT_WHICH_CAN_BE_HELD_IN_A_SINT THEN
	RETURN;
END_IF

IF in < DatatypeLimits.MIN_VALUE_OF_DINT_WHICH_CAN_BE_HELD_IN_A_SINT THEN
	RETURN;
END_IF

out := DINT_TO_SINT(in);
TryConvert_DINT_TO_SINT := TRUE;

END_FUNCTION

// Converters/DINT_TO_/TryConvert_DINT_TO_INT
FUNCTION TryConvert_DINT_TO_INT : BOOL
VAR_INPUT
	in : DINT;
	out : REFERENCE TO INT;
END_VAR

IF in > DatatypeLimits.MAX_VALUE_OF_DINT_WHICH_CAN_BE_HELD_IN_A_INT THEN
	RETURN;
END_IF

IF in < DatatypeLimits.MIN_VALUE_OF_DINT_WHICH_CAN_BE_HELD_IN_A_INT THEN
	RETURN;
END_IF

out := DINT_TO_INT(in);
TryConvert_DINT_TO_INT := TRUE;

END_FUNCTION

// Converters/DINT_TO_/TryConvert_DINT_TO_DINT
FUNCTION TryConvert_DINT_TO_DINT : BOOL
VAR_INPUT
	in : DINT;
	out : REFERENCE TO DINT;
END_VAR

out := in;
TryConvert_DINT_TO_DINT := TRUE;

END_FUNCTION

// Converters/DINT_TO_/TryConvert_DINT_TO_LINT
FUNCTION TryConvert_DINT_TO_LINT : BOOL
VAR_INPUT
	in : DINT;
	out : REFERENCE TO LINT;
END_VAR

out := DINT_TO_LINT(in);
TryConvert_DINT_TO_LINT := TRUE;

END_FUNCTION

// Converters/DINT_TO_/TryConvert_DINT_TO_USINT
FUNCTION TryConvert_DINT_TO_USINT : BOOL
VAR_INPUT
	in : DINT;
	out : REFERENCE TO USINT;
END_VAR

IF in > DatatypeLimits.MAX_VALUE_OF_DINT_WHICH_CAN_BE_HELD_IN_A_USINT THEN
	RETURN;
END_IF

IF in < DatatypeLimits.MIN_VALUE_OF_DINT_WHICH_CAN_BE_HELD_IN_A_USINT THEN
	RETURN;
END_IF

out := DINT_TO_USINT(in);
TryConvert_DINT_TO_USINT := TRUE;

END_FUNCTION

// Converters/DINT_TO_/TryConvert_DINT_TO_UINT
FUNCTION TryConvert_DINT_TO_UINT : BOOL
VAR_INPUT
	in : DINT;
	out : REFERENCE TO UINT;
END_VAR

IF in > DatatypeLimits.MAX_VALUE_OF_DINT_WHICH_CAN_BE_HELD_IN_A_UINT THEN
	RETURN;
END_IF

IF in < DatatypeLimits.MIN_VALUE_OF_DINT_WHICH_CAN_BE_HELD_IN_A_UINT THEN
	RETURN;
END_IF

out := DINT_TO_UINT(in);
TryConvert_DINT_TO_UINT := TRUE;

END_FUNCTION

// Converters/DINT_TO_/TryConvert_DINT_TO_UDINT
FUNCTION TryConvert_DINT_TO_UDINT : BOOL
VAR_INPUT
	in : DINT;
	out : REFERENCE TO UDINT;
END_VAR

IF in < DatatypeLimits.MIN_VALUE_OF_DINT_WHICH_CAN_BE_HELD_IN_A_UDINT THEN
	RETURN;
END_IF

out := DINT_TO_UDINT(in);
TryConvert_DINT_TO_UDINT := TRUE;

END_FUNCTION

// Converters/DINT_TO_/TryConvert_DINT_TO_ULINT
FUNCTION TryConvert_DINT_TO_ULINT : BOOL
VAR_INPUT
	in : DINT;
	out : REFERENCE TO ULINT;
END_VAR

IF in < DatatypeLimits.MIN_VALUE_OF_DINT_WHICH_CAN_BE_HELD_IN_A_ULINT THEN
	RETURN;
END_IF

out := DINT_TO_ULINT(in);
TryConvert_DINT_TO_ULINT := TRUE;

END_FUNCTION

// Converters/DINT_TO_/TryConvert_DINT_TO_REAL
FUNCTION TryConvert_DINT_TO_REAL : BOOL
VAR_INPUT
	in : DINT;
	out : REFERENCE TO REAL;
END_VAR

out := DINT_TO_REAL(in);
TryConvert_DINT_TO_REAL := TRUE;

END_FUNCTION

// Converters/DINT_TO_/TryConvert_DINT_TO_LREAL
FUNCTION TryConvert_DINT_TO_LREAL : BOOL
VAR_INPUT
	in : DINT;
	out : REFERENCE TO LREAL;
END_VAR

out := DINT_TO_LREAL(in);
TryConvert_DINT_TO_LREAL := TRUE;

END_FUNCTION

// Converters/DINT_TO_/TryConvert_DINT_TO_TIME
FUNCTION TryConvert_DINT_TO_TIME : BOOL
VAR_INPUT
	in : DINT;
	out : REFERENCE TO TIME;
END_VAR

IF in < DatatypeLimits.MIN_VALUE_OF_DINT_WHICH_CAN_BE_HELD_IN_A_TIME THEN
	RETURN;
END_IF

out := DINT_TO_TIME(in);
TryConvert_DINT_TO_TIME := TRUE;

END_FUNCTION

// Converters/DINT_TO_/TryConvert_DINT_TO_TOD
FUNCTION TryConvert_DINT_TO_TOD : BOOL
VAR_INPUT
	in : DINT;
	out : REFERENCE TO TOD;
END_VAR

IF in > DatatypeLimits.MAX_VALUE_OF_DINT_WHICH_CAN_BE_HELD_IN_A_TOD THEN
	RETURN;
END_IF

IF in < DatatypeLimits.MIN_VALUE_OF_DINT_WHICH_CAN_BE_HELD_IN_A_TOD THEN
	RETURN;
END_IF

out := DINT_TO_TOD(in);
TryConvert_DINT_TO_TOD := TRUE;

END_FUNCTION

// Converters/DINT_TO_/TryConvert_DINT_TO_DT
FUNCTION TryConvert_DINT_TO_DT : BOOL
VAR_INPUT
	in : DINT;
	out : REFERENCE TO DT;
END_VAR

IF in < DatatypeLimits.MIN_VALUE_OF_DINT_WHICH_CAN_BE_HELD_IN_A_DT THEN
	RETURN;
END_IF

out := DINT_TO_DT(in);
TryConvert_DINT_TO_DT := TRUE;

END_FUNCTION

// Converters/DINT_TO_/TryConvert_DINT_TO_STRING
FUNCTION TryConvert_DINT_TO_STRING : BOOL
VAR_INPUT
	in : DINT;
	out : REFERENCE TO STRING;
END_VAR

out := DINT_TO_STRING(in);
TryConvert_DINT_TO_STRING := TRUE;

END_FUNCTION

// Converters/DT_TO_/TryConvert_DT_TO_BOOL
FUNCTION TryConvert_DT_TO_BOOL : BOOL
VAR_INPUT
	in : DT;
	out : REFERENCE TO BOOL;
END_VAR

out := DT_TO_BOOL(in);
TryConvert_DT_TO_BOOL := TRUE;

END_FUNCTION

// Converters/DT_TO_/TryConvert_DT_TO_BYTE
FUNCTION TryConvert_DT_TO_BYTE : BOOL
VAR_INPUT
	in : DT;
	out : REFERENCE TO BYTE;
END_VAR

IF in > DatatypeLimits.MAX_VALUE_OF_DT_WHICH_CAN_BE_HELD_IN_A_BYTE THEN
	RETURN;
END_IF

out := DT_TO_BYTE(in);
TryConvert_DT_TO_BYTE := TRUE;

END_FUNCTION

// Converters/DT_TO_/TryConvert_DT_TO_DATE
FUNCTION TryConvert_DT_TO_DATE : BOOL
VAR_INPUT
	in : DT;
	out : REFERENCE TO DATE;
END_VAR

out := DT_TO_DATE(in);
TryConvert_DT_TO_DATE := TRUE;

END_FUNCTION

// Converters/DT_TO_/TryConvert_DT_TO_Destination
FUNCTION TryConvert_DT_TO_Destination : BOOL
VAR_INPUT
	in : DT;
	out : ANY;
END_VAR
VAR
	convertResult : BOOL := FALSE;
	convertAddress : PVOID;
	_BOOL : BOOL;
	_BYTE : BYTE;
	_WORD : WORD;
	_DWORD : DWORD;
	_LWORD : LWORD;
	_SINT : SINT;
	_INT : INT;
	_DINT : DINT;
	_LINT : LINT;
	_USINT : USINT;
	_UINT : UINT;
	_UDINT : UDINT;
	_ULINT : ULINT;
	_REAL : REAL;
	_LREAL : LREAL;
	_TIME : TIME;
	_TOD : TOD;
	_DATE : DATE;
	_DT : DT;
	_STRING : STRING;
END_VAR

CASE out.TypeClass OF
	__SYSTEM.TYPE_CLASS.TYPE_BOOL:
	
	convertResult := TryConvert_DT_TO_BOOL(in, _BOOL);
	IF convertResult THEN
		convertAddress := ADR(_BOOL);
	END_IF
	
	__SYSTEM.TYPE_CLASS.TYPE_BYTE:
	
	convertResult := TryConvert_DT_TO_BYTE(in, _BYTE);
	IF convertResult THEN
		convertAddress := ADR(_BYTE);
	END_IF
	
	__SYSTEM.TYPE_CLASS.TYPE_WORD:
	
	convertResult := TryConvert_DT_TO_WORD(in, _WORD);
	IF convertResult THEN
		convertAddress := ADR(_WORD);
	END_IF
	
	__SYSTEM.TYPE_CLASS.TYPE_DWORD:
	
	convertResult := TryConvert_DT_TO_DWORD(in, _DWORD);
	IF convertResult THEN
		convertAddress := ADR(_DWORD);
	END_IF
	
	__SYSTEM.TYPE_CLASS.TYPE_LWORD:
	
	convertResult := TryConvert_DT_TO_LWORD(in, _LWORD);
	IF convertResult THEN
		convertAddress := ADR(_LWORD);
	END_IF
	
	__SYSTEM.TYPE_CLASS.TYPE_SINT:
	
	convertResult := TryConvert_DT_TO_SINT(in, _SINT);
	IF convertResult THEN
		convertAddress := ADR(_SINT);
	END_IF
	
	__SYSTEM.TYPE_CLASS.TYPE_INT:
	
	convertResult := TryConvert_DT_TO_INT(in, _INT);
	IF convertResult THEN
		convertAddress := ADR(_INT);
	END_IF
	
	__SYSTEM.TYPE_CLASS.TYPE_DINT:
	
	convertResult := TryConvert_DT_TO_DINT(in, _DINT);
	IF convertResult THEN
		convertAddress := ADR(_DINT);
	END_IF
	
	__SYSTEM.TYPE_CLASS.TYPE_LINT:
	
	convertResult := TryConvert_DT_TO_LINT(in, _LINT);
	IF convertResult THEN
		convertAddress := ADR(_LINT);
	END_IF
	
	__SYSTEM.TYPE_CLASS.TYPE_USINT:
	
	convertResult := TryConvert_DT_TO_USINT(in, _USINT);
	IF convertResult THEN
		convertAddress := ADR(_USINT);
	END_IF
	
	__SYSTEM.TYPE_CLASS.TYPE_UINT:
	
	convertResult := TryConvert_DT_TO_UINT(in, _UINT);
	IF convertResult THEN
		convertAddress := ADR(_UINT);
	END_IF
	
	__SYSTEM.TYPE_CLASS.TYPE_UDINT:
	
	convertResult := TryConvert_DT_TO_UDINT(in, _UDINT);
	IF convertResult THEN
		convertAddress := ADR(_UDINT);
	END_IF
	
	__SYSTEM.TYPE_CLASS.TYPE_ULINT:
	
	convertResult := TryConvert_DT_TO_ULINT(in, _ULINT);
	IF convertResult THEN
		convertAddress := ADR(_ULINT);
	END_IF
	
	__SYSTEM.TYPE_CLASS.TYPE_REAL:
	
	convertResult := TryConvert_DT_TO_REAL(in, _REAL);
	IF convertResult THEN
		convertAddress := ADR(_REAL);
	END_IF
	
	__SYSTEM.TYPE_CLASS.TYPE_LREAL:
	
	convertResult := TryConvert_DT_TO_LREAL(in, _LREAL);
	IF convertResult THEN
		convertAddress := ADR(_LREAL);
	END_IF
	
	__SYSTEM.TYPE_CLASS.TYPE_TIME:
	
	convertResult := TryConvert_DT_TO_TIME(in, _TIME);
	IF convertResult THEN
		convertAddress := ADR(_TIME);
	END_IF
	
	__SYSTEM.TYPE_CLASS.TYPE_TIMEOFDAY:
	
	convertResult := TryConvert_DT_TO_TOD(in, _TOD);
	IF convertResult THEN
		convertAddress := ADR(_TOD);
	END_IF
	
	__SYSTEM.TYPE_CLASS.TYPE_DATE:
	
	convertResult := TryConvert_DT_TO_DATE(in, _DATE);
	IF convertResult THEN
		convertAddress := ADR(_DATE);
	END_IF
	
	__SYSTEM.TYPE_CLASS.TYPE_DATEANDTIME:
	
	convertResult := TryConvert_DT_TO_DT(in, _DT);
	IF convertResult THEN
		convertAddress := ADR(_DT);
	END_IF
	
	__SYSTEM.TYPE_CLASS.TYPE_STRING:
	
	convertResult := TryConvert_DT_TO_STRING(in, _STRING);
	IF convertResult THEN
		convertAddress := ADR(_STRING);
	END_IF
	
END_CASE

IF convertResult THEN
	memcpy(out.pValue,convertAddress,DINT_TO_UDINT(out.diSize));
END_IF

TryConvert_DT_TO_Destination := convertResult;

END_FUNCTION

// Converters/DT_TO_/TryConvert_DT_TO_WORD
FUNCTION TryConvert_DT_TO_WORD : BOOL
VAR_INPUT
	in : DT;
	out : REFERENCE TO WORD;
END_VAR

IF in > DatatypeLimits.MAX_VALUE_OF_DT_WHICH_CAN_BE_HELD_IN_A_WORD THEN
	RETURN;
END_IF

out := DT_TO_WORD(in);
TryConvert_DT_TO_WORD := TRUE;

END_FUNCTION

// Converters/DT_TO_/TryConvert_DT_TO_DWORD
FUNCTION TryConvert_DT_TO_DWORD : BOOL
VAR_INPUT
	in : DT;
	out : REFERENCE TO DWORD;
END_VAR

out := DT_TO_DWORD(in);
TryConvert_DT_TO_DWORD := TRUE;

END_FUNCTION

// Converters/DT_TO_/TryConvert_DT_TO_LWORD
FUNCTION TryConvert_DT_TO_LWORD : BOOL
VAR_INPUT
	in : DT;
	out : REFERENCE TO LWORD;
END_VAR

out := DT_TO_LWORD(in);
TryConvert_DT_TO_LWORD := TRUE;

END_FUNCTION

// Converters/DT_TO_/TryConvert_DT_TO_SINT
FUNCTION TryConvert_DT_TO_SINT : BOOL
VAR_INPUT
	in : DT;
	out : REFERENCE TO SINT;
END_VAR

IF in > DatatypeLimits.MAX_VALUE_OF_DT_WHICH_CAN_BE_HELD_IN_A_SINT THEN
	RETURN;
END_IF

out := DT_TO_SINT(in);
TryConvert_DT_TO_SINT := TRUE;

END_FUNCTION

// Converters/DT_TO_/TryConvert_DT_TO_INT
FUNCTION TryConvert_DT_TO_INT : BOOL
VAR_INPUT
	in : DT;
	out : REFERENCE TO INT;
END_VAR

IF in > DatatypeLimits.MAX_VALUE_OF_DT_WHICH_CAN_BE_HELD_IN_A_INT THEN
	RETURN;
END_IF

out := DT_TO_INT(in);
TryConvert_DT_TO_INT := TRUE;

END_FUNCTION

// Converters/DT_TO_/TryConvert_DT_TO_DINT
FUNCTION TryConvert_DT_TO_DINT : BOOL
VAR_INPUT
	in : DT;
	out : REFERENCE TO DINT;
END_VAR

IF in > DatatypeLimits.MAX_VALUE_OF_DT_WHICH_CAN_BE_HELD_IN_A_DINT THEN
	RETURN;
END_IF

out := DT_TO_DINT(in);
TryConvert_DT_TO_DINT := TRUE;

END_FUNCTION

// Converters/DT_TO_/TryConvert_DT_TO_LINT
FUNCTION TryConvert_DT_TO_LINT : BOOL
VAR_INPUT
	in : DT;
	out : REFERENCE TO LINT;
END_VAR

out := DT_TO_LINT(in);
TryConvert_DT_TO_LINT := TRUE;

END_FUNCTION

// Converters/DT_TO_/TryConvert_DT_TO_USINT
FUNCTION TryConvert_DT_TO_USINT : BOOL
VAR_INPUT
	in : DT;
	out : REFERENCE TO USINT;
END_VAR

IF in > DatatypeLimits.MAX_VALUE_OF_DT_WHICH_CAN_BE_HELD_IN_A_USINT THEN
	RETURN;
END_IF

out := DT_TO_USINT(in);
TryConvert_DT_TO_USINT := TRUE;

END_FUNCTION

// Converters/DT_TO_/TryConvert_DT_TO_UINT
FUNCTION TryConvert_DT_TO_UINT : BOOL
VAR_INPUT
	in : DT;
	out : REFERENCE TO UINT;
END_VAR

IF in > DatatypeLimits.MAX_VALUE_OF_DT_WHICH_CAN_BE_HELD_IN_A_UINT THEN
	RETURN;
END_IF

out := DT_TO_UINT(in);
TryConvert_DT_TO_UINT := TRUE;

END_FUNCTION

// Converters/DT_TO_/TryConvert_DT_TO_UDINT
FUNCTION TryConvert_DT_TO_UDINT : BOOL
VAR_INPUT
	in : DT;
	out : REFERENCE TO UDINT;
END_VAR

out := DT_TO_UDINT(in);
TryConvert_DT_TO_UDINT := TRUE;

END_FUNCTION

// Converters/DT_TO_/TryConvert_DT_TO_ULINT
FUNCTION TryConvert_DT_TO_ULINT : BOOL
VAR_INPUT
	in : DT;
	out : REFERENCE TO ULINT;
END_VAR

out := DT_TO_ULINT(in);
TryConvert_DT_TO_ULINT := TRUE;

END_FUNCTION

// Converters/DT_TO_/TryConvert_DT_TO_REAL
FUNCTION TryConvert_DT_TO_REAL : BOOL
VAR_INPUT
	in : DT;
	out : REFERENCE TO REAL;
END_VAR

out := DT_TO_REAL(in);
TryConvert_DT_TO_REAL := TRUE;

END_FUNCTION

// Converters/DT_TO_/TryConvert_DT_TO_LREAL
FUNCTION TryConvert_DT_TO_LREAL : BOOL
VAR_INPUT
	in : DT;
	out : REFERENCE TO LREAL;
END_VAR

out := DT_TO_LREAL(in);
TryConvert_DT_TO_LREAL := TRUE;

END_FUNCTION

// Converters/DT_TO_/TryConvert_DT_TO_TIME
FUNCTION TryConvert_DT_TO_TIME : BOOL
VAR_INPUT
	in : DT;
	out : REFERENCE TO TIME;
END_VAR

IF in > DatatypeLimits.MAX_VALUE_OF_DT_WHICH_CAN_BE_HELD_IN_A_TIME THEN
	RETURN;
END_IF

out := DT_TO_TIME(in);
TryConvert_DT_TO_TIME := TRUE;

END_FUNCTION

// Converters/DT_TO_/TryConvert_DT_TO_TOD
FUNCTION TryConvert_DT_TO_TOD : BOOL
VAR_INPUT
	in : DT;
	out : REFERENCE TO TOD;
END_VAR

IF in > DatatypeLimits.MAX_VALUE_OF_DT_WHICH_CAN_BE_HELD_IN_A_TOD THEN
	RETURN;
END_IF

out := DT_TO_TOD(in);
TryConvert_DT_TO_TOD := TRUE;

END_FUNCTION

// Converters/DT_TO_/TryConvert_DT_TO_DT
FUNCTION TryConvert_DT_TO_DT : BOOL
VAR_INPUT
	in : DT;
	out : REFERENCE TO DT;
END_VAR

out := in;
TryConvert_DT_TO_DT := TRUE;

END_FUNCTION

// Converters/DT_TO_/TryConvert_DT_TO_STRING
FUNCTION TryConvert_DT_TO_STRING : BOOL
VAR_INPUT
	in : DT;
	out : REFERENCE TO STRING;
END_VAR

out := DT_TO_STRING(in);
TryConvert_DT_TO_STRING := TRUE;

END_FUNCTION

// Converters/DWORD_TO_/TryConvert_DWORD_TO_BOOL
FUNCTION TryConvert_DWORD_TO_BOOL : BOOL
VAR_INPUT
	in : DWORD;
	out : REFERENCE TO BOOL;
END_VAR

out := DWORD_TO_BOOL(in);
TryConvert_DWORD_TO_BOOL := TRUE;

END_FUNCTION

// Converters/DWORD_TO_/TryConvert_DWORD_TO_BYTE
FUNCTION TryConvert_DWORD_TO_BYTE : BOOL
VAR_INPUT
	in : DWORD;
	out : REFERENCE TO BYTE;
END_VAR

IF in > DatatypeLimits.MAX_VALUE_OF_DWORD_WHICH_CAN_BE_HELD_IN_A_BYTE THEN
	RETURN;
END_IF

out := DWORD_TO_BYTE(in);
TryConvert_DWORD_TO_BYTE := TRUE;

END_FUNCTION

// Converters/DWORD_TO_/TryConvert_DWORD_TO_DATE
FUNCTION TryConvert_DWORD_TO_DATE : BOOL
VAR_INPUT
	in : DWORD;
	out : REFERENCE TO DATE;
END_VAR

out := DWORD_TO_DATE(in);
TryConvert_DWORD_TO_DATE := TRUE;

END_FUNCTION

// Converters/DWORD_TO_/TryConvert_DWORD_TO_Destination
FUNCTION TryConvert_DWORD_TO_Destination : BOOL
VAR_INPUT
	in : DWORD;
	out : ANY;
END_VAR
VAR
	convertResult : BOOL := FALSE;
	convertAddress : PVOID;
	_BOOL : BOOL;
	_BYTE : BYTE;
	_WORD : WORD;
	_DWORD : DWORD;
	_LWORD : LWORD;
	_SINT : SINT;
	_INT : INT;
	_DINT : DINT;
	_LINT : LINT;
	_USINT : USINT;
	_UINT : UINT;
	_UDINT : UDINT;
	_ULINT : ULINT;
	_REAL : REAL;
	_LREAL : LREAL;
	_TIME : TIME;
	_TOD : TOD;
	_DATE : DATE;
	_DT : DT;
	_STRING : STRING;
END_VAR

CASE out.TypeClass OF
	__SYSTEM.TYPE_CLASS.TYPE_BOOL:
	
	convertResult := TryConvert_DWORD_TO_BOOL(in, _BOOL);
	IF convertResult THEN
		convertAddress := ADR(_BOOL);
	END_IF
	
	__SYSTEM.TYPE_CLASS.TYPE_BYTE:
	
	convertResult := TryConvert_DWORD_TO_BYTE(in, _BYTE);
	IF convertResult THEN
		convertAddress := ADR(_BYTE);
	END_IF
	
	__SYSTEM.TYPE_CLASS.TYPE_WORD:
	
	convertResult := TryConvert_DWORD_TO_WORD(in, _WORD);
	IF convertResult THEN
		convertAddress := ADR(_WORD);
	END_IF
	
	__SYSTEM.TYPE_CLASS.TYPE_DWORD:
	
	convertResult := TryConvert_DWORD_TO_DWORD(in, _DWORD);
	IF convertResult THEN
		convertAddress := ADR(_DWORD);
	END_IF
	
	__SYSTEM.TYPE_CLASS.TYPE_LWORD:
	
	convertResult := TryConvert_DWORD_TO_LWORD(in, _LWORD);
	IF convertResult THEN
		convertAddress := ADR(_LWORD);
	END_IF
	
	__SYSTEM.TYPE_CLASS.TYPE_SINT:
	
	convertResult := TryConvert_DWORD_TO_SINT(in, _SINT);
	IF convertResult THEN
		convertAddress := ADR(_SINT);
	END_IF
	
	__SYSTEM.TYPE_CLASS.TYPE_INT:
	
	convertResult := TryConvert_DWORD_TO_INT(in, _INT);
	IF convertResult THEN
		convertAddress := ADR(_INT);
	END_IF
	
	__SYSTEM.TYPE_CLASS.TYPE_DINT:
	
	convertResult := TryConvert_DWORD_TO_DINT(in, _DINT);
	IF convertResult THEN
		convertAddress := ADR(_DINT);
	END_IF
	
	__SYSTEM.TYPE_CLASS.TYPE_LINT:
	
	convertResult := TryConvert_DWORD_TO_LINT(in, _LINT);
	IF convertResult THEN
		convertAddress := ADR(_LINT);
	END_IF
	
	__SYSTEM.TYPE_CLASS.TYPE_USINT:
	
	convertResult := TryConvert_DWORD_TO_USINT(in, _USINT);
	IF convertResult THEN
		convertAddress := ADR(_USINT);
	END_IF
	
	__SYSTEM.TYPE_CLASS.TYPE_UINT:
	
	convertResult := TryConvert_DWORD_TO_UINT(in, _UINT);
	IF convertResult THEN
		convertAddress := ADR(_UINT);
	END_IF
	
	__SYSTEM.TYPE_CLASS.TYPE_UDINT:
	
	convertResult := TryConvert_DWORD_TO_UDINT(in, _UDINT);
	IF convertResult THEN
		convertAddress := ADR(_UDINT);
	END_IF
	
	__SYSTEM.TYPE_CLASS.TYPE_ULINT:
	
	convertResult := TryConvert_DWORD_TO_ULINT(in, _ULINT);
	IF convertResult THEN
		convertAddress := ADR(_ULINT);
	END_IF
	
	__SYSTEM.TYPE_CLASS.TYPE_REAL:
	
	convertResult := TryConvert_DWORD_TO_REAL(in, _REAL);
	IF convertResult THEN
		convertAddress := ADR(_REAL);
	END_IF
	
	__SYSTEM.TYPE_CLASS.TYPE_LREAL:
	
	convertResult := TryConvert_DWORD_TO_LREAL(in, _LREAL);
	IF convertResult THEN
		convertAddress := ADR(_LREAL);
	END_IF
	
	__SYSTEM.TYPE_CLASS.TYPE_TIME:
	
	convertResult := TryConvert_DWORD_TO_TIME(in, _TIME);
	IF convertResult THEN
		convertAddress := ADR(_TIME);
	END_IF
	
	__SYSTEM.TYPE_CLASS.TYPE_TIMEOFDAY:
	
	convertResult := TryConvert_DWORD_TO_TOD(in, _TOD);
	IF convertResult THEN
		convertAddress := ADR(_TOD);
	END_IF
	
	__SYSTEM.TYPE_CLASS.TYPE_DATE:
	
	convertResult := TryConvert_DWORD_TO_DATE(in, _DATE);
	IF convertResult THEN
		convertAddress := ADR(_DATE);
	END_IF
	
	__SYSTEM.TYPE_CLASS.TYPE_DATEANDTIME:
	
	convertResult := TryConvert_DWORD_TO_DT(in, _DT);
	IF convertResult THEN
		convertAddress := ADR(_DT);
	END_IF
	
	__SYSTEM.TYPE_CLASS.TYPE_STRING:
	
	convertResult := TryConvert_DWORD_TO_STRING(in, _STRING);
	IF convertResult THEN
		convertAddress := ADR(_STRING);
	END_IF
	
END_CASE

IF convertResult THEN
	memcpy(out.pValue,convertAddress,DINT_TO_UDINT(out.diSize));
END_IF

TryConvert_DWORD_TO_Destination := convertResult;

END_FUNCTION

// Converters/DWORD_TO_/TryConvert_DWORD_TO_WORD
FUNCTION TryConvert_DWORD_TO_WORD : BOOL
VAR_INPUT
	in : DWORD;
	out : REFERENCE TO WORD;
END_VAR

IF in > DatatypeLimits.MAX_VALUE_OF_DWORD_WHICH_CAN_BE_HELD_IN_A_WORD THEN
	RETURN;
END_IF

out := DWORD_TO_WORD(in);
TryConvert_DWORD_TO_WORD := TRUE;

END_FUNCTION

// Converters/DWORD_TO_/TryConvert_DWORD_TO_DWORD
FUNCTION TryConvert_DWORD_TO_DWORD : BOOL
VAR_INPUT
	in : DWORD;
	out : REFERENCE TO DWORD;
END_VAR

out := in;
TryConvert_DWORD_TO_DWORD := TRUE;

END_FUNCTION

// Converters/DWORD_TO_/TryConvert_DWORD_TO_LWORD
FUNCTION TryConvert_DWORD_TO_LWORD : BOOL
VAR_INPUT
	in : DWORD;
	out : REFERENCE TO LWORD;
END_VAR

out := DWORD_TO_LWORD(in);
TryConvert_DWORD_TO_LWORD := TRUE;

END_FUNCTION

// Converters/DWORD_TO_/TryConvert_DWORD_TO_SINT
FUNCTION TryConvert_DWORD_TO_SINT : BOOL
VAR_INPUT
	in : DWORD;
	out : REFERENCE TO SINT;
END_VAR

IF in > DatatypeLimits.MAX_VALUE_OF_DWORD_WHICH_CAN_BE_HELD_IN_A_SINT THEN
	RETURN;
END_IF

out := DWORD_TO_SINT(in);
TryConvert_DWORD_TO_SINT := TRUE;

END_FUNCTION

// Converters/DWORD_TO_/TryConvert_DWORD_TO_INT
FUNCTION TryConvert_DWORD_TO_INT : BOOL
VAR_INPUT
	in : DWORD;
	out : REFERENCE TO INT;
END_VAR

IF in > DatatypeLimits.MAX_VALUE_OF_DWORD_WHICH_CAN_BE_HELD_IN_A_INT THEN
	RETURN;
END_IF

out := DWORD_TO_INT(in);
TryConvert_DWORD_TO_INT := TRUE;

END_FUNCTION

// Converters/DWORD_TO_/TryConvert_DWORD_TO_DINT
FUNCTION TryConvert_DWORD_TO_DINT : BOOL
VAR_INPUT
	in : DWORD;
	out : REFERENCE TO DINT;
END_VAR

IF in > DatatypeLimits.MAX_VALUE_OF_DWORD_WHICH_CAN_BE_HELD_IN_A_DINT THEN
	RETURN;
END_IF

out := DWORD_TO_DINT(in);
TryConvert_DWORD_TO_DINT := TRUE;

END_FUNCTION

// Converters/DWORD_TO_/TryConvert_DWORD_TO_LINT
FUNCTION TryConvert_DWORD_TO_LINT : BOOL
VAR_INPUT
	in : DWORD;
	out : REFERENCE TO LINT;
END_VAR

out := DWORD_TO_LINT(in);
TryConvert_DWORD_TO_LINT := TRUE;

END_FUNCTION

// Converters/DWORD_TO_/TryConvert_DWORD_TO_USINT
FUNCTION TryConvert_DWORD_TO_USINT : BOOL
VAR_INPUT
	in : DWORD;
	out : REFERENCE TO USINT;
END_VAR

IF in > DatatypeLimits.MAX_VALUE_OF_DWORD_WHICH_CAN_BE_HELD_IN_A_USINT THEN
	RETURN;
END_IF

out := DWORD_TO_USINT(in);
TryConvert_DWORD_TO_USINT := TRUE;

END_FUNCTION

// Converters/DWORD_TO_/TryConvert_DWORD_TO_UINT
FUNCTION TryConvert_DWORD_TO_UINT : BOOL
VAR_INPUT
	in : DWORD;
	out : REFERENCE TO UINT;
END_VAR

IF in > DatatypeLimits.MAX_VALUE_OF_DWORD_WHICH_CAN_BE_HELD_IN_A_UINT THEN
	RETURN;
END_IF

out := DWORD_TO_UINT(in);
TryConvert_DWORD_TO_UINT := TRUE;

END_FUNCTION

// Converters/DWORD_TO_/TryConvert_DWORD_TO_UDINT
FUNCTION TryConvert_DWORD_TO_UDINT : BOOL
VAR_INPUT
	in : DWORD;
	out : REFERENCE TO UDINT;
END_VAR

out := DWORD_TO_UDINT(in);
TryConvert_DWORD_TO_UDINT := TRUE;

END_FUNCTION

// Converters/DWORD_TO_/TryConvert_DWORD_TO_ULINT
FUNCTION TryConvert_DWORD_TO_ULINT : BOOL
VAR_INPUT
	in : DWORD;
	out : REFERENCE TO ULINT;
END_VAR

out := DWORD_TO_ULINT(in);
TryConvert_DWORD_TO_ULINT := TRUE;

END_FUNCTION

// Converters/DWORD_TO_/TryConvert_DWORD_TO_REAL
FUNCTION TryConvert_DWORD_TO_REAL : BOOL
VAR_INPUT
	in : DWORD;
	out : REFERENCE TO REAL;
END_VAR

out := DWORD_TO_REAL(in);
TryConvert_DWORD_TO_REAL := TRUE;

END_FUNCTION

// Converters/DWORD_TO_/TryConvert_DWORD_TO_LREAL
FUNCTION TryConvert_DWORD_TO_LREAL : BOOL
VAR_INPUT
	in : DWORD;
	out : REFERENCE TO LREAL;
END_VAR

out := DWORD_TO_LREAL(in);
TryConvert_DWORD_TO_LREAL := TRUE;

END_FUNCTION

// Converters/DWORD_TO_/TryConvert_DWORD_TO_TIME
FUNCTION TryConvert_DWORD_TO_TIME : BOOL
VAR_INPUT
	in : DWORD;
	out : REFERENCE TO TIME;
END_VAR

out := DWORD_TO_TIME(in);
TryConvert_DWORD_TO_TIME := TRUE;

END_FUNCTION

// Converters/DWORD_TO_/TryConvert_DWORD_TO_TOD
FUNCTION TryConvert_DWORD_TO_TOD : BOOL
VAR_INPUT
	in : DWORD;
	out : REFERENCE TO TOD;
END_VAR

IF in > DatatypeLimits.MAX_VALUE_OF_DWORD_WHICH_CAN_BE_HELD_IN_A_TOD THEN
	RETURN;
END_IF

out := DWORD_TO_TOD(in);
TryConvert_DWORD_TO_TOD := TRUE;

END_FUNCTION

// Converters/DWORD_TO_/TryConvert_DWORD_TO_DT
FUNCTION TryConvert_DWORD_TO_DT : BOOL
VAR_INPUT
	in : DWORD;
	out : REFERENCE TO DT;
END_VAR

out := DWORD_TO_DT(in);
TryConvert_DWORD_TO_DT := TRUE;

END_FUNCTION

// Converters/DWORD_TO_/TryConvert_DWORD_TO_STRING
FUNCTION TryConvert_DWORD_TO_STRING : BOOL
VAR_INPUT
	in : DWORD;
	out : REFERENCE TO STRING;
END_VAR

out := DWORD_TO_STRING(in);
TryConvert_DWORD_TO_STRING := TRUE;

END_FUNCTION

// Converters/INT_TO_/TryConvert_INT_TO_BOOL
FUNCTION TryConvert_INT_TO_BOOL : BOOL
VAR_INPUT
	in : INT;
	out : REFERENCE TO BOOL;
END_VAR

out := INT_TO_BOOL(in);
TryConvert_INT_TO_BOOL := TRUE;

END_FUNCTION

// Converters/INT_TO_/TryConvert_INT_TO_BYTE
FUNCTION TryConvert_INT_TO_BYTE : BOOL
VAR_INPUT
	in : INT;
	out : REFERENCE TO BYTE;
END_VAR

IF in > DatatypeLimits.MAX_VALUE_OF_INT_WHICH_CAN_BE_HELD_IN_A_BYTE THEN
	RETURN;
END_IF

IF in < DatatypeLimits.MIN_VALUE_OF_INT_WHICH_CAN_BE_HELD_IN_A_BYTE THEN
	RETURN;
END_IF

out := INT_TO_BYTE(in);
TryConvert_INT_TO_BYTE := TRUE;

END_FUNCTION

// Converters/INT_TO_/TryConvert_INT_TO_DATE
FUNCTION TryConvert_INT_TO_DATE : BOOL
VAR_INPUT
	in : INT;
	out : REFERENCE TO DATE;
END_VAR

IF in < DatatypeLimits.MIN_VALUE_OF_INT_WHICH_CAN_BE_HELD_IN_A_DATE THEN
	RETURN;
END_IF

out := INT_TO_DATE(in);
TryConvert_INT_TO_DATE := TRUE;

END_FUNCTION

// Converters/INT_TO_/TryConvert_INT_TO_Destination
FUNCTION TryConvert_INT_TO_Destination : BOOL
VAR_INPUT
	in : INT;
	out : ANY;
END_VAR
VAR
	convertResult : BOOL := FALSE;
	convertAddress : PVOID;
	_BOOL : BOOL;
	_BYTE : BYTE;
	_WORD : WORD;
	_DWORD : DWORD;
	_LWORD : LWORD;
	_SINT : SINT;
	_INT : INT;
	_DINT : DINT;
	_LINT : LINT;
	_USINT : USINT;
	_UINT : UINT;
	_UDINT : UDINT;
	_ULINT : ULINT;
	_REAL : REAL;
	_LREAL : LREAL;
	_TIME : TIME;
	_TOD : TOD;
	_DATE : DATE;
	_DT : DT;
	_STRING : STRING;
END_VAR

CASE out.TypeClass OF
	__SYSTEM.TYPE_CLASS.TYPE_BOOL:
	
	convertResult := TryConvert_INT_TO_BOOL(in, _BOOL);
	IF convertResult THEN
		convertAddress := ADR(_BOOL);
	END_IF
	
	__SYSTEM.TYPE_CLASS.TYPE_BYTE:
	
	convertResult := TryConvert_INT_TO_BYTE(in, _BYTE);
	IF convertResult THEN
		convertAddress := ADR(_BYTE);
	END_IF
	
	__SYSTEM.TYPE_CLASS.TYPE_WORD:
	
	convertResult := TryConvert_INT_TO_WORD(in, _WORD);
	IF convertResult THEN
		convertAddress := ADR(_WORD);
	END_IF
	
	__SYSTEM.TYPE_CLASS.TYPE_DWORD:
	
	convertResult := TryConvert_INT_TO_DWORD(in, _DWORD);
	IF convertResult THEN
		convertAddress := ADR(_DWORD);
	END_IF
	
	__SYSTEM.TYPE_CLASS.TYPE_LWORD:
	
	convertResult := TryConvert_INT_TO_LWORD(in, _LWORD);
	IF convertResult THEN
		convertAddress := ADR(_LWORD);
	END_IF
	
	__SYSTEM.TYPE_CLASS.TYPE_SINT:
	
	convertResult := TryConvert_INT_TO_SINT(in, _SINT);
	IF convertResult THEN
		convertAddress := ADR(_SINT);
	END_IF
	
	__SYSTEM.TYPE_CLASS.TYPE_INT:
	
	convertResult := TryConvert_INT_TO_INT(in, _INT);
	IF convertResult THEN
		convertAddress := ADR(_INT);
	END_IF
	
	__SYSTEM.TYPE_CLASS.TYPE_DINT:
	
	convertResult := TryConvert_INT_TO_DINT(in, _DINT);
	IF convertResult THEN
		convertAddress := ADR(_DINT);
	END_IF
	
	__SYSTEM.TYPE_CLASS.TYPE_LINT:
	
	convertResult := TryConvert_INT_TO_LINT(in, _LINT);
	IF convertResult THEN
		convertAddress := ADR(_LINT);
	END_IF
	
	__SYSTEM.TYPE_CLASS.TYPE_USINT:
	
	convertResult := TryConvert_INT_TO_USINT(in, _USINT);
	IF convertResult THEN
		convertAddress := ADR(_USINT);
	END_IF
	
	__SYSTEM.TYPE_CLASS.TYPE_UINT:
	
	convertResult := TryConvert_INT_TO_UINT(in, _UINT);
	IF convertResult THEN
		convertAddress := ADR(_UINT);
	END_IF
	
	__SYSTEM.TYPE_CLASS.TYPE_UDINT:
	
	convertResult := TryConvert_INT_TO_UDINT(in, _UDINT);
	IF convertResult THEN
		convertAddress := ADR(_UDINT);
	END_IF
	
	__SYSTEM.TYPE_CLASS.TYPE_ULINT:
	
	convertResult := TryConvert_INT_TO_ULINT(in, _ULINT);
	IF convertResult THEN
		convertAddress := ADR(_ULINT);
	END_IF
	
	__SYSTEM.TYPE_CLASS.TYPE_REAL:
	
	convertResult := TryConvert_INT_TO_REAL(in, _REAL);
	IF convertResult THEN
		convertAddress := ADR(_REAL);
	END_IF
	
	__SYSTEM.TYPE_CLASS.TYPE_LREAL:
	
	convertResult := TryConvert_INT_TO_LREAL(in, _LREAL);
	IF convertResult THEN
		convertAddress := ADR(_LREAL);
	END_IF
	
	__SYSTEM.TYPE_CLASS.TYPE_TIME:
	
	convertResult := TryConvert_INT_TO_TIME(in, _TIME);
	IF convertResult THEN
		convertAddress := ADR(_TIME);
	END_IF
	
	__SYSTEM.TYPE_CLASS.TYPE_TIMEOFDAY:
	
	convertResult := TryConvert_INT_TO_TOD(in, _TOD);
	IF convertResult THEN
		convertAddress := ADR(_TOD);
	END_IF
	
	__SYSTEM.TYPE_CLASS.TYPE_DATE:
	
	convertResult := TryConvert_INT_TO_DATE(in, _DATE);
	IF convertResult THEN
		convertAddress := ADR(_DATE);
	END_IF
	
	__SYSTEM.TYPE_CLASS.TYPE_DATEANDTIME:
	
	convertResult := TryConvert_INT_TO_DT(in, _DT);
	IF convertResult THEN
		convertAddress := ADR(_DT);
	END_IF
	
	__SYSTEM.TYPE_CLASS.TYPE_STRING:
	
	convertResult := TryConvert_INT_TO_STRING(in, _STRING);
	IF convertResult THEN
		convertAddress := ADR(_STRING);
	END_IF
	
END_CASE

IF convertResult THEN
	memcpy(out.pValue,convertAddress,DINT_TO_UDINT(out.diSize));
END_IF

TryConvert_INT_TO_Destination := convertResult;

END_FUNCTION

// Converters/INT_TO_/TryConvert_INT_TO_WORD
FUNCTION TryConvert_INT_TO_WORD : BOOL
VAR_INPUT
	in : INT;
	out : REFERENCE TO WORD;
END_VAR

IF in < DatatypeLimits.MIN_VALUE_OF_INT_WHICH_CAN_BE_HELD_IN_A_WORD THEN
	RETURN;
END_IF

out := INT_TO_WORD(in);
TryConvert_INT_TO_WORD := TRUE;

END_FUNCTION

// Converters/INT_TO_/TryConvert_INT_TO_DWORD
FUNCTION TryConvert_INT_TO_DWORD : BOOL
VAR_INPUT
	in : INT;
	out : REFERENCE TO DWORD;
END_VAR

IF in < DatatypeLimits.MIN_VALUE_OF_INT_WHICH_CAN_BE_HELD_IN_A_DWORD THEN
	RETURN;
END_IF

out := INT_TO_DWORD(in);
TryConvert_INT_TO_DWORD := TRUE;

END_FUNCTION

// Converters/INT_TO_/TryConvert_INT_TO_LWORD
FUNCTION TryConvert_INT_TO_LWORD : BOOL
VAR_INPUT
	in : INT;
	out : REFERENCE TO LWORD;
END_VAR

IF in < DatatypeLimits.MIN_VALUE_OF_INT_WHICH_CAN_BE_HELD_IN_A_LWORD THEN
	RETURN;
END_IF

out := INT_TO_LWORD(in);
TryConvert_INT_TO_LWORD := TRUE;

END_FUNCTION

// Converters/INT_TO_/TryConvert_INT_TO_SINT
FUNCTION TryConvert_INT_TO_SINT : BOOL
VAR_INPUT
	in : INT;
	out : REFERENCE TO SINT;
END_VAR

IF in > DatatypeLimits.MAX_VALUE_OF_INT_WHICH_CAN_BE_HELD_IN_A_SINT THEN
	RETURN;
END_IF

IF in < DatatypeLimits.MIN_VALUE_OF_INT_WHICH_CAN_BE_HELD_IN_A_SINT THEN
	RETURN;
END_IF

out := INT_TO_SINT(in);
TryConvert_INT_TO_SINT := TRUE;

END_FUNCTION

// Converters/INT_TO_/TryConvert_INT_TO_INT
FUNCTION TryConvert_INT_TO_INT : BOOL
VAR_INPUT
	in : INT;
	out : REFERENCE TO INT;
END_VAR

out := in;
TryConvert_INT_TO_INT := TRUE;

END_FUNCTION

// Converters/INT_TO_/TryConvert_INT_TO_DINT
FUNCTION TryConvert_INT_TO_DINT : BOOL
VAR_INPUT
	in : INT;
	out : REFERENCE TO DINT;
END_VAR

out := INT_TO_DINT(in);
TryConvert_INT_TO_DINT := TRUE;

END_FUNCTION

// Converters/INT_TO_/TryConvert_INT_TO_LINT
FUNCTION TryConvert_INT_TO_LINT : BOOL
VAR_INPUT
	in : INT;
	out : REFERENCE TO LINT;
END_VAR

out := INT_TO_LINT(in);
TryConvert_INT_TO_LINT := TRUE;

END_FUNCTION

// Converters/INT_TO_/TryConvert_INT_TO_USINT
FUNCTION TryConvert_INT_TO_USINT : BOOL
VAR_INPUT
	in : INT;
	out : REFERENCE TO USINT;
END_VAR

IF in > DatatypeLimits.MAX_VALUE_OF_INT_WHICH_CAN_BE_HELD_IN_A_USINT THEN
	RETURN;
END_IF

IF in < DatatypeLimits.MIN_VALUE_OF_INT_WHICH_CAN_BE_HELD_IN_A_USINT THEN
	RETURN;
END_IF

out := INT_TO_USINT(in);
TryConvert_INT_TO_USINT := TRUE;

END_FUNCTION

// Converters/INT_TO_/TryConvert_INT_TO_UINT
FUNCTION TryConvert_INT_TO_UINT : BOOL
VAR_INPUT
	in : INT;
	out : REFERENCE TO UINT;
END_VAR

IF in < DatatypeLimits.MIN_VALUE_OF_INT_WHICH_CAN_BE_HELD_IN_A_UINT THEN
	RETURN;
END_IF

out := INT_TO_UINT(in);
TryConvert_INT_TO_UINT := TRUE;

END_FUNCTION

// Converters/INT_TO_/TryConvert_INT_TO_UDINT
FUNCTION TryConvert_INT_TO_UDINT : BOOL
VAR_INPUT
	in : INT;
	out : REFERENCE TO UDINT;
END_VAR

IF in < DatatypeLimits.MIN_VALUE_OF_INT_WHICH_CAN_BE_HELD_IN_A_UDINT THEN
	RETURN;
END_IF

out := INT_TO_UDINT(in);
TryConvert_INT_TO_UDINT := TRUE;

END_FUNCTION

// Converters/INT_TO_/TryConvert_INT_TO_ULINT
FUNCTION TryConvert_INT_TO_ULINT : BOOL
VAR_INPUT
	in : INT;
	out : REFERENCE TO ULINT;
END_VAR

IF in < DatatypeLimits.MIN_VALUE_OF_INT_WHICH_CAN_BE_HELD_IN_A_ULINT THEN
	RETURN;
END_IF

out := INT_TO_ULINT(in);
TryConvert_INT_TO_ULINT := TRUE;

END_FUNCTION

// Converters/INT_TO_/TryConvert_INT_TO_REAL
FUNCTION TryConvert_INT_TO_REAL : BOOL
VAR_INPUT
	in : INT;
	out : REFERENCE TO REAL;
END_VAR

out := INT_TO_REAL(in);
TryConvert_INT_TO_REAL := TRUE;

END_FUNCTION

// Converters/INT_TO_/TryConvert_INT_TO_LREAL
FUNCTION TryConvert_INT_TO_LREAL : BOOL
VAR_INPUT
	in : INT;
	out : REFERENCE TO LREAL;
END_VAR

out := INT_TO_LREAL(in);
TryConvert_INT_TO_LREAL := TRUE;

END_FUNCTION

// Converters/INT_TO_/TryConvert_INT_TO_TIME
FUNCTION TryConvert_INT_TO_TIME : BOOL
VAR_INPUT
	in : INT;
	out : REFERENCE TO TIME;
END_VAR

IF in < DatatypeLimits.MIN_VALUE_OF_INT_WHICH_CAN_BE_HELD_IN_A_TIME THEN
	RETURN;
END_IF

out := INT_TO_TIME(in);
TryConvert_INT_TO_TIME := TRUE;

END_FUNCTION

// Converters/INT_TO_/TryConvert_INT_TO_TOD
FUNCTION TryConvert_INT_TO_TOD : BOOL
VAR_INPUT
	in : INT;
	out : REFERENCE TO TOD;
END_VAR

IF in < DatatypeLimits.MIN_VALUE_OF_INT_WHICH_CAN_BE_HELD_IN_A_TOD THEN
	RETURN;
END_IF

out := INT_TO_TOD(in);
TryConvert_INT_TO_TOD := TRUE;

END_FUNCTION

// Converters/INT_TO_/TryConvert_INT_TO_DT
FUNCTION TryConvert_INT_TO_DT : BOOL
VAR_INPUT
	in : INT;
	out : REFERENCE TO DT;
END_VAR

IF in < DatatypeLimits.MIN_VALUE_OF_INT_WHICH_CAN_BE_HELD_IN_A_DT THEN
	RETURN;
END_IF

out := INT_TO_DT(in);
TryConvert_INT_TO_DT := TRUE;

END_FUNCTION

// Converters/INT_TO_/TryConvert_INT_TO_STRING
FUNCTION TryConvert_INT_TO_STRING : BOOL
VAR_INPUT
	in : INT;
	out : REFERENCE TO STRING;
END_VAR

out := INT_TO_STRING(in);
TryConvert_INT_TO_STRING := TRUE;

END_FUNCTION

// Converters/LINT_TO_/TryConvert_LINT_TO_BOOL
FUNCTION TryConvert_LINT_TO_BOOL : BOOL
VAR_INPUT
	in : LINT;
	out : REFERENCE TO BOOL;
END_VAR

out := LINT_TO_BOOL(in);
TryConvert_LINT_TO_BOOL := TRUE;

END_FUNCTION

// Converters/LINT_TO_/TryConvert_LINT_TO_BYTE
FUNCTION TryConvert_LINT_TO_BYTE : BOOL
VAR_INPUT
	in : LINT;
	out : REFERENCE TO BYTE;
END_VAR

IF in > DatatypeLimits.MAX_VALUE_OF_LINT_WHICH_CAN_BE_HELD_IN_A_BYTE THEN
	RETURN;
END_IF

IF in < DatatypeLimits.MIN_VALUE_OF_LINT_WHICH_CAN_BE_HELD_IN_A_BYTE THEN
	RETURN;
END_IF

out := LINT_TO_BYTE(in);
TryConvert_LINT_TO_BYTE := TRUE;

END_FUNCTION

// Converters/LINT_TO_/TryConvert_LINT_TO_DATE
FUNCTION TryConvert_LINT_TO_DATE : BOOL
VAR_INPUT
	in : LINT;
	out : REFERENCE TO DATE;
END_VAR

IF in > DatatypeLimits.MAX_VALUE_OF_LINT_WHICH_CAN_BE_HELD_IN_A_DATE THEN
	RETURN;
END_IF

IF in < DatatypeLimits.MIN_VALUE_OF_LINT_WHICH_CAN_BE_HELD_IN_A_DATE THEN
	RETURN;
END_IF

out := LINT_TO_DATE(in);
TryConvert_LINT_TO_DATE := TRUE;

END_FUNCTION

// Converters/LINT_TO_/TryConvert_LINT_TO_Destination
FUNCTION TryConvert_LINT_TO_Destination : BOOL
VAR_INPUT
	in : LINT;
	out : ANY;
END_VAR
VAR
	convertResult : BOOL := FALSE;
	convertAddress : PVOID;
	_BOOL : BOOL;
	_BYTE : BYTE;
	_WORD : WORD;
	_DWORD : DWORD;
	_LWORD : LWORD;
	_SINT : SINT;
	_INT : INT;
	_DINT : DINT;
	_LINT : LINT;
	_USINT : USINT;
	_UINT : UINT;
	_UDINT : UDINT;
	_ULINT : ULINT;
	_REAL : REAL;
	_LREAL : LREAL;
	_TIME : TIME;
	_TOD : TOD;
	_DATE : DATE;
	_DT : DT;
	_STRING : STRING;
END_VAR

CASE out.TypeClass OF
	__SYSTEM.TYPE_CLASS.TYPE_BOOL:
	
	convertResult := TryConvert_LINT_TO_BOOL(in, _BOOL);
	IF convertResult THEN
		convertAddress := ADR(_BOOL);
	END_IF
	
	__SYSTEM.TYPE_CLASS.TYPE_BYTE:
	
	convertResult := TryConvert_LINT_TO_BYTE(in, _BYTE);
	IF convertResult THEN
		convertAddress := ADR(_BYTE);
	END_IF
	
	__SYSTEM.TYPE_CLASS.TYPE_WORD:
	
	convertResult := TryConvert_LINT_TO_WORD(in, _WORD);
	IF convertResult THEN
		convertAddress := ADR(_WORD);
	END_IF
	
	__SYSTEM.TYPE_CLASS.TYPE_DWORD:
	
	convertResult := TryConvert_LINT_TO_DWORD(in, _DWORD);
	IF convertResult THEN
		convertAddress := ADR(_DWORD);
	END_IF
	
	__SYSTEM.TYPE_CLASS.TYPE_LWORD:
	
	convertResult := TryConvert_LINT_TO_LWORD(in, _LWORD);
	IF convertResult THEN
		convertAddress := ADR(_LWORD);
	END_IF
	
	__SYSTEM.TYPE_CLASS.TYPE_SINT:
	
	convertResult := TryConvert_LINT_TO_SINT(in, _SINT);
	IF convertResult THEN
		convertAddress := ADR(_SINT);
	END_IF
	
	__SYSTEM.TYPE_CLASS.TYPE_INT:
	
	convertResult := TryConvert_LINT_TO_INT(in, _INT);
	IF convertResult THEN
		convertAddress := ADR(_INT);
	END_IF
	
	__SYSTEM.TYPE_CLASS.TYPE_DINT:
	
	convertResult := TryConvert_LINT_TO_DINT(in, _DINT);
	IF convertResult THEN
		convertAddress := ADR(_DINT);
	END_IF
	
	__SYSTEM.TYPE_CLASS.TYPE_LINT:
	
	convertResult := TryConvert_LINT_TO_LINT(in, _LINT);
	IF convertResult THEN
		convertAddress := ADR(_LINT);
	END_IF
	
	__SYSTEM.TYPE_CLASS.TYPE_USINT:
	
	convertResult := TryConvert_LINT_TO_USINT(in, _USINT);
	IF convertResult THEN
		convertAddress := ADR(_USINT);
	END_IF
	
	__SYSTEM.TYPE_CLASS.TYPE_UINT:
	
	convertResult := TryConvert_LINT_TO_UINT(in, _UINT);
	IF convertResult THEN
		convertAddress := ADR(_UINT);
	END_IF
	
	__SYSTEM.TYPE_CLASS.TYPE_UDINT:
	
	convertResult := TryConvert_LINT_TO_UDINT(in, _UDINT);
	IF convertResult THEN
		convertAddress := ADR(_UDINT);
	END_IF
	
	__SYSTEM.TYPE_CLASS.TYPE_ULINT:
	
	convertResult := TryConvert_LINT_TO_ULINT(in, _ULINT);
	IF convertResult THEN
		convertAddress := ADR(_ULINT);
	END_IF
	
	__SYSTEM.TYPE_CLASS.TYPE_REAL:
	
	convertResult := TryConvert_LINT_TO_REAL(in, _REAL);
	IF convertResult THEN
		convertAddress := ADR(_REAL);
	END_IF
	
	__SYSTEM.TYPE_CLASS.TYPE_LREAL:
	
	convertResult := TryConvert_LINT_TO_LREAL(in, _LREAL);
	IF convertResult THEN
		convertAddress := ADR(_LREAL);
	END_IF
	
	__SYSTEM.TYPE_CLASS.TYPE_TIME:
	
	convertResult := TryConvert_LINT_TO_TIME(in, _TIME);
	IF convertResult THEN
		convertAddress := ADR(_TIME);
	END_IF
	
	__SYSTEM.TYPE_CLASS.TYPE_TIMEOFDAY:
	
	convertResult := TryConvert_LINT_TO_TOD(in, _TOD);
	IF convertResult THEN
		convertAddress := ADR(_TOD);
	END_IF
	
	__SYSTEM.TYPE_CLASS.TYPE_DATE:
	
	convertResult := TryConvert_LINT_TO_DATE(in, _DATE);
	IF convertResult THEN
		convertAddress := ADR(_DATE);
	END_IF
	
	__SYSTEM.TYPE_CLASS.TYPE_DATEANDTIME:
	
	convertResult := TryConvert_LINT_TO_DT(in, _DT);
	IF convertResult THEN
		convertAddress := ADR(_DT);
	END_IF
	
	__SYSTEM.TYPE_CLASS.TYPE_STRING:
	
	convertResult := TryConvert_LINT_TO_STRING(in, _STRING);
	IF convertResult THEN
		convertAddress := ADR(_STRING);
	END_IF
	
END_CASE

IF convertResult THEN
	memcpy(out.pValue,convertAddress,DINT_TO_UDINT(out.diSize));
END_IF

TryConvert_LINT_TO_Destination := convertResult;

END_FUNCTION

// Converters/LINT_TO_/TryConvert_LINT_TO_WORD
FUNCTION TryConvert_LINT_TO_WORD : BOOL
VAR_INPUT
	in : LINT;
	out : REFERENCE TO WORD;
END_VAR

IF in > DatatypeLimits.MAX_VALUE_OF_LINT_WHICH_CAN_BE_HELD_IN_A_WORD THEN
	RETURN;
END_IF

IF in < DatatypeLimits.MIN_VALUE_OF_LINT_WHICH_CAN_BE_HELD_IN_A_WORD THEN
	RETURN;
END_IF

out := LINT_TO_WORD(in);
TryConvert_LINT_TO_WORD := TRUE;

END_FUNCTION

// Converters/LINT_TO_/TryConvert_LINT_TO_DWORD
FUNCTION TryConvert_LINT_TO_DWORD : BOOL
VAR_INPUT
	in : LINT;
	out : REFERENCE TO DWORD;
END_VAR

IF in > DatatypeLimits.MAX_VALUE_OF_LINT_WHICH_CAN_BE_HELD_IN_A_DWORD THEN
	RETURN;
END_IF

IF in < DatatypeLimits.MIN_VALUE_OF_LINT_WHICH_CAN_BE_HELD_IN_A_DWORD THEN
	RETURN;
END_IF

out := LINT_TO_DWORD(in);
TryConvert_LINT_TO_DWORD := TRUE;

END_FUNCTION

// Converters/LINT_TO_/TryConvert_LINT_TO_LWORD
FUNCTION TryConvert_LINT_TO_LWORD : BOOL
VAR_INPUT
	in : LINT;
	out : REFERENCE TO LWORD;
END_VAR

IF in < DatatypeLimits.MIN_VALUE_OF_LINT_WHICH_CAN_BE_HELD_IN_A_LWORD THEN
	RETURN;
END_IF

out := LINT_TO_LWORD(in);
TryConvert_LINT_TO_LWORD := TRUE;

END_FUNCTION

// Converters/LINT_TO_/TryConvert_LINT_TO_SINT
FUNCTION TryConvert_LINT_TO_SINT : BOOL
VAR_INPUT
	in : LINT;
	out : REFERENCE TO SINT;
END_VAR

IF in > DatatypeLimits.MAX_VALUE_OF_LINT_WHICH_CAN_BE_HELD_IN_A_SINT THEN
	RETURN;
END_IF

IF in < DatatypeLimits.MIN_VALUE_OF_LINT_WHICH_CAN_BE_HELD_IN_A_SINT THEN
	RETURN;
END_IF

out := LINT_TO_SINT(in);
TryConvert_LINT_TO_SINT := TRUE;

END_FUNCTION

// Converters/LINT_TO_/TryConvert_LINT_TO_INT
FUNCTION TryConvert_LINT_TO_INT : BOOL
VAR_INPUT
	in : LINT;
	out : REFERENCE TO INT;
END_VAR

IF in > DatatypeLimits.MAX_VALUE_OF_LINT_WHICH_CAN_BE_HELD_IN_A_INT THEN
	RETURN;
END_IF

IF in < DatatypeLimits.MIN_VALUE_OF_LINT_WHICH_CAN_BE_HELD_IN_A_INT THEN
	RETURN;
END_IF

out := LINT_TO_INT(in);
TryConvert_LINT_TO_INT := TRUE;

END_FUNCTION

// Converters/LINT_TO_/TryConvert_LINT_TO_DINT
FUNCTION TryConvert_LINT_TO_DINT : BOOL
VAR_INPUT
	in : LINT;
	out : REFERENCE TO DINT;
END_VAR

IF in > DatatypeLimits.MAX_VALUE_OF_LINT_WHICH_CAN_BE_HELD_IN_A_DINT THEN
	RETURN;
END_IF

IF in < DatatypeLimits.MIN_VALUE_OF_LINT_WHICH_CAN_BE_HELD_IN_A_DINT THEN
	RETURN;
END_IF

out := LINT_TO_DINT(in);
TryConvert_LINT_TO_DINT := TRUE;

END_FUNCTION

// Converters/LINT_TO_/TryConvert_LINT_TO_LINT
FUNCTION TryConvert_LINT_TO_LINT : BOOL
VAR_INPUT
	in : LINT;
	out : REFERENCE TO LINT;
END_VAR

out := in;
TryConvert_LINT_TO_LINT := TRUE;

END_FUNCTION

// Converters/LINT_TO_/TryConvert_LINT_TO_USINT
FUNCTION TryConvert_LINT_TO_USINT : BOOL
VAR_INPUT
	in : LINT;
	out : REFERENCE TO USINT;
END_VAR

IF in > DatatypeLimits.MAX_VALUE_OF_LINT_WHICH_CAN_BE_HELD_IN_A_USINT THEN
	RETURN;
END_IF

IF in < DatatypeLimits.MIN_VALUE_OF_LINT_WHICH_CAN_BE_HELD_IN_A_USINT THEN
	RETURN;
END_IF

out := LINT_TO_USINT(in);
TryConvert_LINT_TO_USINT := TRUE;

END_FUNCTION

// Converters/LINT_TO_/TryConvert_LINT_TO_UINT
FUNCTION TryConvert_LINT_TO_UINT : BOOL
VAR_INPUT
	in : LINT;
	out : REFERENCE TO UINT;
END_VAR

IF in > DatatypeLimits.MAX_VALUE_OF_LINT_WHICH_CAN_BE_HELD_IN_A_UINT THEN
	RETURN;
END_IF

IF in < DatatypeLimits.MIN_VALUE_OF_LINT_WHICH_CAN_BE_HELD_IN_A_UINT THEN
	RETURN;
END_IF

out := LINT_TO_UINT(in);
TryConvert_LINT_TO_UINT := TRUE;

END_FUNCTION

// Converters/LINT_TO_/TryConvert_LINT_TO_UDINT
FUNCTION TryConvert_LINT_TO_UDINT : BOOL
VAR_INPUT
	in : LINT;
	out : REFERENCE TO UDINT;
END_VAR

IF in > DatatypeLimits.MAX_VALUE_OF_LINT_WHICH_CAN_BE_HELD_IN_A_UDINT THEN
	RETURN;
END_IF

IF in < DatatypeLimits.MIN_VALUE_OF_LINT_WHICH_CAN_BE_HELD_IN_A_UDINT THEN
	RETURN;
END_IF

out := LINT_TO_UDINT(in);
TryConvert_LINT_TO_UDINT := TRUE;

END_FUNCTION

// Converters/LINT_TO_/TryConvert_LINT_TO_ULINT
FUNCTION TryConvert_LINT_TO_ULINT : BOOL
VAR_INPUT
	in : LINT;
	out : REFERENCE TO ULINT;
END_VAR

IF in < DatatypeLimits.MIN_VALUE_OF_LINT_WHICH_CAN_BE_HELD_IN_A_ULINT THEN
	RETURN;
END_IF

out := LINT_TO_ULINT(in);
TryConvert_LINT_TO_ULINT := TRUE;

END_FUNCTION

// Converters/LINT_TO_/TryConvert_LINT_TO_REAL
FUNCTION TryConvert_LINT_TO_REAL : BOOL
VAR_INPUT
	in : LINT;
	out : REFERENCE TO REAL;
END_VAR

out := LINT_TO_REAL(in);
TryConvert_LINT_TO_REAL := TRUE;

END_FUNCTION

// Converters/LINT_TO_/TryConvert_LINT_TO_LREAL
FUNCTION TryConvert_LINT_TO_LREAL : BOOL
VAR_INPUT
	in : LINT;
	out : REFERENCE TO LREAL;
END_VAR

out := LINT_TO_LREAL(in);
TryConvert_LINT_TO_LREAL := TRUE;

END_FUNCTION

// Converters/LINT_TO_/TryConvert_LINT_TO_TIME
FUNCTION TryConvert_LINT_TO_TIME : BOOL
VAR_INPUT
	in : LINT;
	out : REFERENCE TO TIME;
END_VAR

IF in > DatatypeLimits.MAX_VALUE_OF_LINT_WHICH_CAN_BE_HELD_IN_A_TIME THEN
	RETURN;
END_IF

IF in < DatatypeLimits.MIN_VALUE_OF_LINT_WHICH_CAN_BE_HELD_IN_A_TIME THEN
	RETURN;
END_IF

out := LINT_TO_TIME(in);
TryConvert_LINT_TO_TIME := TRUE;

END_FUNCTION

// Converters/LINT_TO_/TryConvert_LINT_TO_TOD
FUNCTION TryConvert_LINT_TO_TOD : BOOL
VAR_INPUT
	in : LINT;
	out : REFERENCE TO TOD;
END_VAR

IF in > DatatypeLimits.MAX_VALUE_OF_LINT_WHICH_CAN_BE_HELD_IN_A_TOD THEN
	RETURN;
END_IF

IF in < DatatypeLimits.MIN_VALUE_OF_LINT_WHICH_CAN_BE_HELD_IN_A_TOD THEN
	RETURN;
END_IF

out := LINT_TO_TOD(in);
TryConvert_LINT_TO_TOD := TRUE;

END_FUNCTION

// Converters/LINT_TO_/TryConvert_LINT_TO_DT
FUNCTION TryConvert_LINT_TO_DT : BOOL
VAR_INPUT
	in : LINT;
	out : REFERENCE TO DT;
END_VAR

IF in > DatatypeLimits.MAX_VALUE_OF_LINT_WHICH_CAN_BE_HELD_IN_A_DT THEN
	RETURN;
END_IF

IF in < DatatypeLimits.MIN_VALUE_OF_LINT_WHICH_CAN_BE_HELD_IN_A_DT THEN
	RETURN;
END_IF

out := LINT_TO_DT(in);
TryConvert_LINT_TO_DT := TRUE;

END_FUNCTION

// Converters/LINT_TO_/TryConvert_LINT_TO_STRING
FUNCTION TryConvert_LINT_TO_STRING : BOOL
VAR_INPUT
	in : LINT;
	out : REFERENCE TO STRING;
END_VAR

out := LINT_TO_STRING(in);
TryConvert_LINT_TO_STRING := TRUE;

END_FUNCTION

// Converters/LREAL_TO_/TryConvert_LREAL_TO_BOOL
FUNCTION TryConvert_LREAL_TO_BOOL : BOOL
VAR_INPUT
	in : LREAL;
	out : REFERENCE TO BOOL;
END_VAR

out := LREAL_TO_BOOL(in);
TryConvert_LREAL_TO_BOOL := TRUE;

END_FUNCTION

// Converters/LREAL_TO_/TryConvert_LREAL_TO_BYTE
FUNCTION TryConvert_LREAL_TO_BYTE : BOOL
VAR_INPUT
	in : LREAL;
	out : REFERENCE TO BYTE;
END_VAR

IF in > DatatypeLimits.MAX_VALUE_OF_LREAL_WHICH_CAN_BE_HELD_IN_A_BYTE THEN
	RETURN;
END_IF

IF in < DatatypeLimits.MIN_VALUE_OF_LREAL_WHICH_CAN_BE_HELD_IN_A_BYTE THEN
	RETURN;
END_IF

out := LREAL_TO_BYTE(in);
TryConvert_LREAL_TO_BYTE := TRUE;

END_FUNCTION

// Converters/LREAL_TO_/TryConvert_LREAL_TO_DATE
FUNCTION TryConvert_LREAL_TO_DATE : BOOL
VAR_INPUT
	in : LREAL;
	out : REFERENCE TO DATE;
END_VAR

IF in > DatatypeLimits.MAX_VALUE_OF_LREAL_WHICH_CAN_BE_HELD_IN_A_DATE THEN
	RETURN;
END_IF

IF in < DatatypeLimits.MIN_VALUE_OF_LREAL_WHICH_CAN_BE_HELD_IN_A_DATE THEN
	RETURN;
END_IF

out := LREAL_TO_DATE(in);
TryConvert_LREAL_TO_DATE := TRUE;

END_FUNCTION

// Converters/LREAL_TO_/TryConvert_LREAL_TO_Destination
FUNCTION TryConvert_LREAL_TO_Destination : BOOL
VAR_INPUT
	in : LREAL;
	out : ANY;
END_VAR
VAR
	convertResult : BOOL := FALSE;
	convertAddress : PVOID;
	_BOOL : BOOL;
	_BYTE : BYTE;
	_WORD : WORD;
	_DWORD : DWORD;
	_LWORD : LWORD;
	_SINT : SINT;
	_INT : INT;
	_DINT : DINT;
	_LINT : LINT;
	_USINT : USINT;
	_UINT : UINT;
	_UDINT : UDINT;
	_ULINT : ULINT;
	_REAL : REAL;
	_LREAL : LREAL;
	_TIME : TIME;
	_TOD : TOD;
	_DATE : DATE;
	_DT : DT;
	_STRING : STRING;
END_VAR

CASE out.TypeClass OF
	__SYSTEM.TYPE_CLASS.TYPE_BOOL:
	
	convertResult := TryConvert_LREAL_TO_BOOL(in, _BOOL);
	IF convertResult THEN
		convertAddress := ADR(_BOOL);
	END_IF
	
	__SYSTEM.TYPE_CLASS.TYPE_BYTE:
	
	convertResult := TryConvert_LREAL_TO_BYTE(in, _BYTE);
	IF convertResult THEN
		convertAddress := ADR(_BYTE);
	END_IF
	
	__SYSTEM.TYPE_CLASS.TYPE_WORD:
	
	convertResult := TryConvert_LREAL_TO_WORD(in, _WORD);
	IF convertResult THEN
		convertAddress := ADR(_WORD);
	END_IF
	
	__SYSTEM.TYPE_CLASS.TYPE_DWORD:
	
	convertResult := TryConvert_LREAL_TO_DWORD(in, _DWORD);
	IF convertResult THEN
		convertAddress := ADR(_DWORD);
	END_IF
	
	__SYSTEM.TYPE_CLASS.TYPE_LWORD:
	
	convertResult := TryConvert_LREAL_TO_LWORD(in, _LWORD);
	IF convertResult THEN
		convertAddress := ADR(_LWORD);
	END_IF
	
	__SYSTEM.TYPE_CLASS.TYPE_SINT:
	
	convertResult := TryConvert_LREAL_TO_SINT(in, _SINT);
	IF convertResult THEN
		convertAddress := ADR(_SINT);
	END_IF
	
	__SYSTEM.TYPE_CLASS.TYPE_INT:
	
	convertResult := TryConvert_LREAL_TO_INT(in, _INT);
	IF convertResult THEN
		convertAddress := ADR(_INT);
	END_IF
	
	__SYSTEM.TYPE_CLASS.TYPE_DINT:
	
	convertResult := TryConvert_LREAL_TO_DINT(in, _DINT);
	IF convertResult THEN
		convertAddress := ADR(_DINT);
	END_IF
	
	__SYSTEM.TYPE_CLASS.TYPE_LINT:
	
	convertResult := TryConvert_LREAL_TO_LINT(in, _LINT);
	IF convertResult THEN
		convertAddress := ADR(_LINT);
	END_IF
	
	__SYSTEM.TYPE_CLASS.TYPE_USINT:
	
	convertResult := TryConvert_LREAL_TO_USINT(in, _USINT);
	IF convertResult THEN
		convertAddress := ADR(_USINT);
	END_IF
	
	__SYSTEM.TYPE_CLASS.TYPE_UINT:
	
	convertResult := TryConvert_LREAL_TO_UINT(in, _UINT);
	IF convertResult THEN
		convertAddress := ADR(_UINT);
	END_IF
	
	__SYSTEM.TYPE_CLASS.TYPE_UDINT:
	
	convertResult := TryConvert_LREAL_TO_UDINT(in, _UDINT);
	IF convertResult THEN
		convertAddress := ADR(_UDINT);
	END_IF
	
	__SYSTEM.TYPE_CLASS.TYPE_ULINT:
	
	convertResult := TryConvert_LREAL_TO_ULINT(in, _ULINT);
	IF convertResult THEN
		convertAddress := ADR(_ULINT);
	END_IF
	
	__SYSTEM.TYPE_CLASS.TYPE_REAL:
	
	convertResult := TryConvert_LREAL_TO_REAL(in, _REAL);
	IF convertResult THEN
		convertAddress := ADR(_REAL);
	END_IF
	
	__SYSTEM.TYPE_CLASS.TYPE_LREAL:
	
	convertResult := TryConvert_LREAL_TO_LREAL(in, _LREAL);
	IF convertResult THEN
		convertAddress := ADR(_LREAL);
	END_IF
	
	__SYSTEM.TYPE_CLASS.TYPE_TIME:
	
	convertResult := TryConvert_LREAL_TO_TIME(in, _TIME);
	IF convertResult THEN
		convertAddress := ADR(_TIME);
	END_IF
	
	__SYSTEM.TYPE_CLASS.TYPE_TIMEOFDAY:
	
	convertResult := TryConvert_LREAL_TO_TOD(in, _TOD);
	IF convertResult THEN
		convertAddress := ADR(_TOD);
	END_IF
	
	__SYSTEM.TYPE_CLASS.TYPE_DATE:
	
	convertResult := TryConvert_LREAL_TO_DATE(in, _DATE);
	IF convertResult THEN
		convertAddress := ADR(_DATE);
	END_IF
	
	__SYSTEM.TYPE_CLASS.TYPE_DATEANDTIME:
	
	convertResult := TryConvert_LREAL_TO_DT(in, _DT);
	IF convertResult THEN
		convertAddress := ADR(_DT);
	END_IF
	
	__SYSTEM.TYPE_CLASS.TYPE_STRING:
	
	convertResult := TryConvert_LREAL_TO_STRING(in, _STRING);
	IF convertResult THEN
		convertAddress := ADR(_STRING);
	END_IF
	
END_CASE

IF convertResult THEN
	memcpy(out.pValue,convertAddress,DINT_TO_UDINT(out.diSize));
END_IF

TryConvert_LREAL_TO_Destination := convertResult;

END_FUNCTION

// Converters/LREAL_TO_/TryConvert_LREAL_TO_WORD
FUNCTION TryConvert_LREAL_TO_WORD : BOOL
VAR_INPUT
	in : LREAL;
	out : REFERENCE TO WORD;
END_VAR

IF in > DatatypeLimits.MAX_VALUE_OF_LREAL_WHICH_CAN_BE_HELD_IN_A_WORD THEN
	RETURN;
END_IF

IF in < DatatypeLimits.MIN_VALUE_OF_LREAL_WHICH_CAN_BE_HELD_IN_A_WORD THEN
	RETURN;
END_IF

out := LREAL_TO_WORD(in);
TryConvert_LREAL_TO_WORD := TRUE;

END_FUNCTION

// Converters/LREAL_TO_/TryConvert_LREAL_TO_DWORD
FUNCTION TryConvert_LREAL_TO_DWORD : BOOL
VAR_INPUT
	in : LREAL;
	out : REFERENCE TO DWORD;
END_VAR

IF in > DatatypeLimits.MAX_VALUE_OF_LREAL_WHICH_CAN_BE_HELD_IN_A_DWORD THEN
	RETURN;
END_IF

IF in < DatatypeLimits.MIN_VALUE_OF_LREAL_WHICH_CAN_BE_HELD_IN_A_DWORD THEN
	RETURN;
END_IF

out := LREAL_TO_DWORD(in);
TryConvert_LREAL_TO_DWORD := TRUE;

END_FUNCTION

// Converters/LREAL_TO_/TryConvert_LREAL_TO_LWORD
FUNCTION TryConvert_LREAL_TO_LWORD : BOOL
VAR_INPUT
	in : LREAL;
	out : REFERENCE TO LWORD;
END_VAR

IF in > DatatypeLimits.MAX_VALUE_OF_LREAL_WHICH_CAN_BE_HELD_IN_A_LWORD THEN
	RETURN;
END_IF

IF in < DatatypeLimits.MIN_VALUE_OF_LREAL_WHICH_CAN_BE_HELD_IN_A_LWORD THEN
	RETURN;
END_IF

out := LREAL_TO_LWORD(in);
TryConvert_LREAL_TO_LWORD := TRUE;

END_FUNCTION

// Converters/LREAL_TO_/TryConvert_LREAL_TO_SINT
FUNCTION TryConvert_LREAL_TO_SINT : BOOL
VAR_INPUT
	in : LREAL;
	out : REFERENCE TO SINT;
END_VAR

IF in > DatatypeLimits.MAX_VALUE_OF_LREAL_WHICH_CAN_BE_HELD_IN_A_SINT THEN
	RETURN;
END_IF

IF in < DatatypeLimits.MIN_VALUE_OF_LREAL_WHICH_CAN_BE_HELD_IN_A_SINT THEN
	RETURN;
END_IF

out := LREAL_TO_SINT(in);
TryConvert_LREAL_TO_SINT := TRUE;

END_FUNCTION

// Converters/LREAL_TO_/TryConvert_LREAL_TO_INT
FUNCTION TryConvert_LREAL_TO_INT : BOOL
VAR_INPUT
	in : LREAL;
	out : REFERENCE TO INT;
END_VAR

IF in > DatatypeLimits.MAX_VALUE_OF_LREAL_WHICH_CAN_BE_HELD_IN_A_INT THEN
	RETURN;
END_IF

IF in < DatatypeLimits.MIN_VALUE_OF_LREAL_WHICH_CAN_BE_HELD_IN_A_INT THEN
	RETURN;
END_IF

out := LREAL_TO_INT(in);
TryConvert_LREAL_TO_INT := TRUE;

END_FUNCTION

// Converters/LREAL_TO_/TryConvert_LREAL_TO_DINT
FUNCTION TryConvert_LREAL_TO_DINT : BOOL
VAR_INPUT
	in : LREAL;
	out : REFERENCE TO DINT;
END_VAR

IF in > DatatypeLimits.MAX_VALUE_OF_LREAL_WHICH_CAN_BE_HELD_IN_A_DINT THEN
	RETURN;
END_IF

